LIN {X 0,Y 149.006,Z 225.633,A -85,B 0,C 180,E1 -24515.4,E2 -24515.4} C_VEL
LIN {X 0,Y 150.508,Z 227.861,A -85,B 0,C 180,E1 -24516.54,E2 -24516.54} C_VEL
LIN {X 0,Y 154.838,Z 237.074,A -85,B 0,C 180,E1 -24520.302,E2 -24520.302} C_VEL
LIN {X 0,Y 156.957,Z 243.18,A -85,B 0,C 180,E1 -24522.459,E2 -24522.459} C_VEL
LIN {X 0,Y 158.651,Z 250.853,A -85,B 0,C 180,E1 -24524.866,E2 -24524.866} C_VEL
LIN {X 0,Y 159.684,Z 260.758,A -85,B 0,C 180,E1 -24527.897,E2 -24527.897} C_VEL
LIN {X 0,Y 159.819,Z 270.245,A -85,B 0,C 180,E1 -24530.92,E2 -24530.92} C_VEL
LIN {X 0,Y 159.177,Z 278.697,A -85,B 0,C 180,E1 -24533.804,E2 -24533.804} C_VEL
LIN {X 0,Y 158.051,Z 285.315,A -85,B 0,C 180,E1 -24536.232,E2 -24536.232} C_VEL
LIN {X 0,Y 154.414,Z 293.15,A -85,B 0,C 180,E1 -24539.201,E2 -24539.201} C_VEL
LIN {X 0,Y 151.168,Z 299.693,A -85,B 0,C 180,E1 -24542.296,E2 -24542.296} C_VEL
LIN {X 0,Y 148.812,Z 304.197,A -85,B 0,C 180,E1 -24544.847,E2 -24544.847} C_VEL
LIN {X 0,Y 145.783,Z 309.692,A -85,B 0,C 180,E1 -24548.804,E2 -24548.804} C_VEL
LIN {X 0,Y 143.391,Z 314.021,A -85,B 0,C 180,E1 -24552.898,E2 -24552.898} C_VEL
LIN {X 0,Y 142.296,Z 316.395,A -85,B 0,C 180,E1 -24555.703,E2 -24555.703} C_VEL
LIN {X 0,Y 141.449,Z 318.201,A -85,B 0,C 180,E1 -24558.537,E2 -24558.537} C_VEL
LIN {X 0,Y 140.623,Z 320.663,A -85,B 0,C 180,E1 -24564.264,E2 -24564.264} C_VEL
LIN {X 0,Y 140.572,Z 321.418,A -85,B 0,C 180,E1 -24569.356,E2 -24569.356} C_VEL
LIN {X 0,Y 140.512,Z 321.259,A -85,B 0,C 180,E1 -24572.867,E2 -24572.867} C_VEL
LIN {X 0,Y 140.624,Z 320.663,A -85,B 0,C 180,E1 -24575.736,E2 -24575.736} C_VEL
LIN {X 0,Y 141.449,Z 318.201,A -85,B 0,C 180,E1 -24581.463,E2 -24581.463} C_VEL
LIN {X 0,Y 142.829,Z 315.242,A -85,B 0,C 180,E1 -24585.702,E2 -24585.702} C_VEL
LIN {X 0,Y 144.913,Z 311.247,A -85,B 0,C 180,E1 -24589.845,E2 -24589.845} C_VEL
LIN {X 0,Y 147.707,Z 306.113,A -85,B 0,C 180,E1 -24593.855,E2 -24593.855} C_VEL
LIN {X 0,Y 150.602,Z 300.85,A -85,B 0,C 180,E1 -24597.064,E2 -24597.064} C_VEL
LIN {X 0,Y 153.725,Z 294.527,A -85,B 0,C 180,E1 -24600.191,E2 -24600.191} C_VEL
LIN {X 0,Y 156.599,Z 288.573,A -85,B 0,C 180,E1 -24602.584,E2 -24602.584} C_VEL
LIN {X 0,Y 158.036,Z 285.315,A -85,B 0,C 180,E1 -24603.771,E2 -24603.771} C_VEL
LIN {X 0,Y 159.42,Z 276.844,A -85,B 0,C 180,E1 -24606.875,E2 -24606.875} C_VEL
LIN {X 0,Y 159.86,Z 266.939,A -85,B 0,C 180,E1 -24610.165,E2 -24610.165} C_VEL
LIN {X 0,Y 159.408,Z 257.125,A -85,B 0,C 180,E1 -24613.205,E2 -24613.205} C_VEL
LIN {X 0,Y 158.142,Z 248.081,A -85,B 0,C 180,E1 -24615.974,E2 -24615.974} C_VEL
LIN {X 0,Y 156.285,Z 240.912,A -85,B 0,C 180,E1 -24618.338,E2 -24618.338} C_VEL
LIN {X 0,Y 154.11,Z 235.491,A -85,B 0,C 180,E1 -24620.322,E2 -24620.322} C_VEL
LIN {X 0,Y 149.931,Z 226.822,A -85,B 0,C 180,E1 -24623.922,E2 -24623.922} C_VEL
LIN {X 0,Y 147.876,Z 223.472,A -85,B 0,C 180,E1 -24625.578,E2 -24625.578} C_VEL
LIN {X 0,Y 147.161,Z 221.537,A -85,B 0,C 180,E1 -24626.317,E2 -24626.317} C_VEL
LIN {X 0,Y 144.734,Z 218.727,A -85,B 0,C 180,E1 -24628.226,E2 -24628.226} C_VEL
LIN {X 0,Y 143.656,Z 215.787,A -85,B 0,C 180,E1 -24629.293,E2 -24629.293} C_VEL
LIN {X 0,Y 143.593,Z 215.404,A -85,B 0,C 180,E1 -24629.491,E2 -24629.491} C_VEL
LIN {X 0,Y 142.834,Z 214.884,A -85,B 0,C 180,E1 -24631.822,E2 -24631.822} C_VEL
LIN {X 0,Y 141.237,Z 214.529,A -85,B 0,C 180,E1 -24634.126,E2 -24634.126} C_VEL
LIN {X 0,Y 136.67,Z 213.808,A -85,B 0,C 180,E1 -24640.471,E2 -24640.471} C_VEL
LIN {X 0,Y 136.278,Z 213.546,A -85,B 0,C 180,E1 -24642.145,E2 -24642.145} C_VEL
LIN {X 0,Y 136.264,Z 213.03,A -85,B 0,C 180,E1 -24645.054,E2 -24645.054} C_VEL
LIN {X 0,Y 136.43,Z 212.991,A -85,B 0,C 180,E1 -24648.165,E2 -24648.165} C_VEL
LIN {X 0,Y 136.55,Z 212.976,A -85,B 0,C 180,E1 -24651.116,E2 -24651.116} C_VEL
LIN {X 0,Y 137.131,Z 212.87,A -85,B 0,C 180,E1 -24659.998,E2 -24659.998} C_VEL
LIN {X 0,Y 136.549,Z 212.968,A -85,B 0,C 180,E1 -24668.881,E2 -24668.881} C_VEL
LIN {X 0,Y 136.438,Z 212.989,A -85,B 0,C 180,E1 -24671.889,E2 -24671.889} C_VEL
LIN {X 0,Y 136.236,Z 213.014,A -85,B 0,C 180,E1 -24678.029,E2 -24678.029} C_VEL
LIN {X 0,Y 136.195,Z 213.016,A -85,B 0,C 180,E1 -24681.747,E2 -24681.747} C_VEL
LIN {X 0,Y 136.083,Z 213.063,A -85,B 0,C 180,E1 -24685.012,E2 -24685.012} C_VEL
LIN {X 0,Y 136.848,Z 215.389,A -85,B 0,C 180,E1 -24686.085,E2 -24686.085} C_VEL
LIN {X 0,Y 138.888,Z 217.815,A -85,B 0,C 180,E1 -24688.3,E2 -24688.3} C_VEL
LIN {X 0,Y 140.193,Z 218.884,A -85,B 0,C 180,E1 -24689.52,E2 -24689.52} C_VEL
LIN {X 0,Y 141.511,Z 221.601,A -85,B 0,C 180,E1 -24691.013,E2 -24691.013} C_VEL
LIN {X 0,Y 143.683,Z 223.961,A -85,B 0,C 180,E1 -24692.892,E2 -24692.892} C_VEL
LIN {X 0,Y 145.775,Z 227.545,A -85,B 0,C 180,E1 -24694.958,E2 -24694.958} C_VEL
LIN {X 0,Y 150.528,Z 235.733,A -85,B 0,C 180,E1 -24699.331,E2 -24699.331} C_VEL
LIN {X 0,Y 154.606,Z 244.364,A -85,B 0,C 180,E1 -24703.339,E2 -24703.339} C_VEL
LIN {X 0,Y 157.554,Z 252.237,A -85,B 0,C 180,E1 -24706.701,E2 -24706.701} C_VEL
LIN {X 0,Y 160.021,Z 261.291,A -85,B 0,C 180,E1 -24710.411,E2 -24710.411} C_VEL
LIN {X 0,Y 161.607,Z 270.196,A -85,B 0,C 180,E1 -24714.119,E2 -24714.119} C_VEL
LIN {X 0,Y 162.565,Z 277.467,A -85,B 0,C 180,E1 -24717.352,E2 -24717.352} C_VEL
LIN {X 0,Y 164.649,Z 285.091,A -85,B 0,C 180,E1 -24721.399,E2 -24721.399} C_VEL
LIN {X 0,Y 167.764,Z 291.175,A -85,B 0,C 180,E1 -24725.234,E2 -24725.234} C_VEL
LIN {X 0,Y 170.94,Z 295.464,A -85,B 0,C 180,E1 -24728.283,E2 -24728.283} C_VEL
LIN {X 0,Y 176.822,Z 300.472,A -85,B 0,C 180,E1 -24732.532,E2 -24732.532} C_VEL
LIN {X 0,Y 184.31,Z 304.617,A -85,B 0,C 180,E1 -24736.774,E2 -24736.774} C_VEL
LIN {X 0,Y 192.385,Z 307.533,A -85,B 0,C 180,E1 -24740.51,E2 -24740.51} C_VEL
LIN {X 0,Y 201.086,Z 309.52,A -85,B 0,C 180,E1 -24743.982,E2 -24743.982} C_VEL
LIN {X 0,Y 206.877,Z 310.378,A -85,B 0,C 180,E1 -24746.104,E2 -24746.104} C_VEL
LIN {X 0,Y 212.302,Z 310.784,A -85,B 0,C 180,E1 -24748.103,E2 -24748.103} C_VEL
LIN {X 0,Y 216.489,Z 310.826,A -85,B 0,C 180,E1 -24750,E2 -24750} C_VEL
LIN {X 0,Y 212.308,Z 310.784,A -85,B 0,C 180,E1 -24751.897,E2 -24751.897} C_VEL
LIN {X 0,Y 204.512,Z 310.094,A -85,B 0,C 180,E1 -24754.756,E2 -24754.756} C_VEL
LIN {X 0,Y 195.226,Z 308.348,A -85,B 0,C 180,E1 -24758.279,E2 -24758.279} C_VEL
LIN {X 0,Y 186.806,Z 305.664,A -85,B 0,C 180,E1 -24762,E2 -24762} C_VEL
LIN {X 0,Y 179.378,Z 302.065,A -85,B 0,C 180,E1 -24765.918,E2 -24765.918} C_VEL
LIN {X 0,Y 173.653,Z 298.041,A -85,B 0,C 180,E1 -24769.595,E2 -24769.595} C_VEL
LIN {X 0,Y 168.814,Z 292.747,A -85,B 0,C 180,E1 -24773.67,E2 -24773.67} C_VEL
LIN {X 0,Y 165.748,Z 287.634,A -85,B 0,C 180,E1 -24777.075,E2 -24777.075} C_VEL
LIN {X 0,Y 163.458,Z 281.287,A -85,B 0,C 180,E1 -24780.696,E2 -24780.696} C_VEL
LIN {X 0,Y 162.202,Z 275.384,A -85,B 0,C 180,E1 -24783.634,E2 -24783.634} C_VEL
LIN {X 0,Y 161.258,Z 267.667,A -85,B 0,C 180,E1 -24786.938,E2 -24786.938} C_VEL
LIN {X 0,Y 159.665,Z 259.89,A -85,B 0,C 180,E1 -24790.157,E2 -24790.157} C_VEL
LIN {X 0,Y 157.138,Z 251.078,A -85,B 0,C 180,E1 -24793.772,E2 -24793.772} C_VEL
LIN {X 0,Y 153.694,Z 242.257,A -85,B 0,C 180,E1 -24797.588,E2 -24797.588} C_VEL
LIN {X 0,Y 149.68,Z 234.222,A -85,B 0,C 180,E1 -24801.464,E2 -24801.464} C_VEL
LIN {X 0,Y 145.781,Z 227.545,A -85,B 0,C 180,E1 -24805.039,E2 -24805.039} C_VEL
LIN {X 0,Y 143.588,Z 223.802,A -85,B 0,C 180,E1 -24807.198,E2 -24807.198} C_VEL
LIN {X 0,Y 141.019,Z 220.798,A -85,B 0,C 180,E1 -24809.49,E2 -24809.49} C_VEL
LIN {X 0,Y 140.07,Z 218.562,A -85,B 0,C 180,E1 -24810.639,E2 -24810.639} C_VEL
LIN {X 0,Y 137.435,Z 216.322,A -85,B 0,C 180,E1 -24813.217,E2 -24813.217} C_VEL
LIN {X 0,Y 136.309,Z 214.128,A -85,B 0,C 180,E1 -24814.624,E2 -24814.624} C_VEL
LIN {X 0,Y 136.084,Z 213.023,A -85,B 0,C 180,E1 -24815.09,E2 -24815.09} C_VEL
LIN {X 0,Y 136.241,Z 213.007,A -85,B 0,C 180,E1 -24818.834,E2 -24818.834} C_VEL
LIN {X 0,Y 136.262,Z 213.001,A -85,B 0,C 180,E1 -24825.057,E2 -24825.057} C_VEL
LIN {X 0,Y 136.429,Z 212.99,A -85,B 0,C 180,E1 -24828.167,E2 -24828.167} C_VEL
LIN {X 0,Y 136.549,Z 212.968,A -85,B 0,C 180,E1 -24831.119,E2 -24831.119} C_VEL
LIN {X 0,Y 137.131,Z 212.87,A -85,B 0,C 180,E1 -24840.002,E2 -24840.002} C_VEL
LIN {X 0,Y 136.55,Z 212.976,A -85,B 0,C 180,E1 -24848.884,E2 -24848.884} C_VEL
LIN {X 0,Y 136.44,Z 212.992,A -85,B 0,C 180,E1 -24851.892,E2 -24851.892} C_VEL
LIN {X 0,Y 136.264,Z 213.031,A -85,B 0,C 180,E1 -24854.946,E2 -24854.946} C_VEL
LIN {X 0,Y 136.387,Z 214.204,A -85,B 0,C 180,E1 -24861.145,E2 -24861.145} C_VEL
LIN {X 0,Y 136.394,Z 215.177,A -85,B 0,C 180,E1 -24865.057,E2 -24865.057} C_VEL
LIN {X 0,Y 137.554,Z 218.297,A -85,B 0,C 180,E1 -24866.557,E2 -24866.557} C_VEL
LIN {X 0,Y 140.111,Z 221.359,A -85,B 0,C 180,E1 -24869.122,E2 -24869.122} C_VEL
LIN {X 0,Y 140.608,Z 222.147,A -85,B 0,C 180,E1 -24869.639,E2 -24869.639} C_VEL
LIN {X 0,Y 142.086,Z 225.426,A -85,B 0,C 180,E1 -24871.291,E2 -24871.291} C_VEL
LIN {X 0,Y 143.909,Z 227.957,A -85,B 0,C 180,E1 -24872.911,E2 -24872.911} C_VEL
LIN {X 0,Y 145.536,Z 231.425,A -85,B 0,C 180,E1 -24874.572,E2 -24874.572} C_VEL
LIN {X 0,Y 146.29,Z 232.543,A -85,B 0,C 180,E1 -24875.245,E2 -24875.245} C_VEL
LIN {X 0,Y 150.351,Z 242.131,A -85,B 0,C 180,E1 -24879.437,E2 -24879.437} C_VEL
LIN {X 0,Y 152.318,Z 249.001,A -85,B 0,C 180,E1 -24881.996,E2 -24881.996} C_VEL
LIN {X 0,Y 153.315,Z 256.047,A -85,B 0,C 180,E1 -24884.384,E2 -24884.384} C_VEL
LIN {X 0,Y 153.814,Z 263.83,A -85,B 0,C 180,E1 -24886.978,E2 -24886.978} C_VEL
LIN {X 0,Y 153.711,Z 271.366,A -85,B 0,C 180,E1 -24889.554,E2 -24889.554} C_VEL
LIN {X 0,Y 153.004,Z 279.042,A -85,B 0,C 180,E1 -24892.339,E2 -24892.339} C_VEL
LIN {X 0,Y 151.946,Z 285.095,A -85,B 0,C 180,E1 -24894.679,E2 -24894.679} C_VEL
LIN {X 0,Y 150.671,Z 288.362,A -85,B 0,C 180,E1 -24895.963,E2 -24895.963} C_VEL
LIN {X 0,Y 147.603,Z 294.315,A -85,B 0,C 180,E1 -24898.416,E2 -24898.416} C_VEL
LIN {X 0,Y 144.259,Z 300.637,A -85,B 0,C 180,E1 -24901.641,E2 -24901.641} C_VEL
LIN {X 0,Y 141.211,Z 305.9,A -85,B 0,C 180,E1 -24904.974,E2 -24904.974} C_VEL
LIN {X 0,Y 138.218,Z 311.034,A -85,B 0,C 180,E1 -24909.15,E2 -24909.15} C_VEL
LIN {X 0,Y 135.96,Z 315.029,A -85,B 0,C 180,E1 -24913.483,E2 -24913.483} C_VEL
LIN {X 0,Y 134.481,Z 317.989,A -85,B 0,C 180,E1 -24917.934,E2 -24917.934} C_VEL
LIN {X 0,Y 133.55,Z 320.452,A -85,B 0,C 180,E1 -24923.959,E2 -24923.959} C_VEL
LIN {X 0,Y 133.415,Z 321.047,A -85,B 0,C 180,E1 -24926.98,E2 -24926.98} C_VEL
LIN {X 0,Y 133.535,Z 321.209,A -85,B 0,C 180,E1 -24930,E2 -24930} C_VEL
LIN {X 0,Y 133.415,Z 321.047,A -85,B 0,C 180,E1 -24933.02,E2 -24933.02} C_VEL
LIN {X 0,Y 133.55,Z 320.452,A -85,B 0,C 180,E1 -24936.041,E2 -24936.041} C_VEL
LIN {X 0,Y 134.481,Z 317.989,A -85,B 0,C 180,E1 -24942.066,E2 -24942.066} C_VEL
LIN {X 0,Y 135.96,Z 315.029,A -85,B 0,C 180,E1 -24946.517,E2 -24946.517} C_VEL
LIN {X 0,Y 138.218,Z 311.034,A -85,B 0,C 180,E1 -24950.85,E2 -24950.85} C_VEL
LIN {X 0,Y 141.213,Z 305.9,A -85,B 0,C 180,E1 -24955.026,E2 -24955.026} C_VEL
LIN {X 0,Y 144.278,Z 300.638,A -85,B 0,C 180,E1 -24958.355,E2 -24958.355} C_VEL
LIN {X 0,Y 146.807,Z 295.829,A -85,B 0,C 180,E1 -24960.892,E2 -24960.892} C_VEL
LIN {X 0,Y 149.855,Z 289.989,A -85,B 0,C 180,E1 -24963.439,E2 -24963.439} C_VEL
LIN {X 0,Y 151.976,Z 285.096,A -85,B 0,C 180,E1 -24965.313,E2 -24965.313} C_VEL
LIN {X 0,Y 153.419,Z 275.912,A -85,B 0,C 180,E1 -24968.851,E2 -24968.851} C_VEL
LIN {X 0,Y 153.842,Z 265.789,A -85,B 0,C 180,E1 -24972.378,E2 -24972.378} C_VEL
LIN {X 0,Y 153.465,Z 257.36,A -85,B 0,C 180,E1 -24975.191,E2 -24975.191} C_VEL
LIN {X 0,Y 152.318,Z 249,A -85,B 0,C 180,E1 -24978.004,E2 -24978.004} C_VEL
LIN {X 0,Y 150.359,Z 242.108,A -85,B 0,C 180,E1 -24980.565,E2 -24980.565} C_VEL
LIN {X 0,Y 146.267,Z 232.458,A -85,B 0,C 180,E1 -24984.787,E2 -24984.787} C_VEL
LIN {X 0,Y 144.221,Z 228.779,A -85,B 0,C 180,E1 -24986.753,E2 -24986.753} C_VEL
LIN {X 0,Y 143.289,Z 226.926,A -85,B 0,C 180,E1 -24987.659,E2 -24987.659} C_VEL
LIN {X 0,Y 141.184,Z 223.799,A -85,B 0,C 180,E1 -24989.629,E2 -24989.629} C_VEL
LIN {X 0,Y 140.238,Z 221.36,A -85,B 0,C 180,E1 -24990.786,E2 -24990.786} C_VEL
LIN {X 0,Y 137.633,Z 218.428,A -85,B 0,C 180,E1 -24993.357,E2 -24993.357} C_VEL
LIN {X 0,Y 136.433,Z 215.428,A -85,B 0,C 180,E1 -24994.849,E2 -24994.849} C_VEL
LIN {X 0,Y 136.356,Z 214.979,A -85,B 0,C 180,E1 -24995.241,E2 -24995.241} C_VEL
LIN {X 0,Y 136.369,Z 214.185,A -85,B 0,C 180,E1 -24998.852,E2 -24998.852} C_VEL
LIN {X 0,Y 136.278,Z 213.546,A -85,B 0,C 180,E1 -25002.145,E2 -25002.145} C_VEL
LIN {X 0,Y 135.512,Z 213.301,A -85,B 0,C 180,E1 -25004.613,E2 -25004.613} C_VEL
LIN {X 0,Y 133.935,Z 213.342,A -85,B 0,C 180,E1 -25007.055,E2 -25007.055} C_VEL
LIN {X 0,Y 129.732,Z 213.826,A -85,B 0,C 180,E1 -25013.797,E2 -25013.797} C_VEL
LIN {X 0,Y 129.544,Z 213.843,A -85,B 0,C 180,E1 -25015.569,E2 -25015.569} C_VEL
LIN {X 0,Y 130.086,Z 213.745,A -85,B 0,C 180,E1 -25019.998,E2 -25019.998} C_VEL
LIN {X 0,Y 129.472,Z 213.847,A -85,B 0,C 180,E1 -25029.37,E2 -25029.37} C_VEL
LIN {X 0,Y 129.342,Z 213.874,A -85,B 0,C 180,E1 -25032.551,E2 -25032.551} C_VEL
LIN {X 0,Y 129.181,Z 213.97,A -85,B 0,C 180,E1 -25037.409,E2 -25037.409} C_VEL
LIN {X 0,Y 129.981,Z 216.424,A -85,B 0,C 180,E1 -25039.133,E2 -25039.133} C_VEL
LIN {X 0,Y 132.512,Z 219.142,A -85,B 0,C 180,E1 -25042.909,E2 -25042.909} C_VEL
LIN {X 0,Y 133.419,Z 219.722,A -85,B 0,C 180,E1 -25043.989,E2 -25043.989} C_VEL
LIN {X 0,Y 134.691,Z 222.539,A -85,B 0,C 180,E1 -25045.911,E2 -25045.911} C_VEL
LIN {X 0,Y 136.26,Z 224.238,A -85,B 0,C 180,E1 -25047.657,E2 -25047.657} C_VEL
LIN {X 0,Y 138.601,Z 227.97,A -85,B 0,C 180,E1 -25050.467,E2 -25050.467} C_VEL
LIN {X 0,Y 139.95,Z 229.469,A -85,B 0,C 180,E1 -25051.821,E2 -25051.821} C_VEL
LIN {X 0,Y 144.323,Z 237.375,A -85,B 0,C 180,E1 -25056.62,E2 -25056.62} C_VEL
LIN {X 0,Y 147.84,Z 244.665,A -85,B 0,C 180,E1 -25060.484,E2 -25060.484} C_VEL
LIN {X 0,Y 150.929,Z 252.576,A -85,B 0,C 180,E1 -25064.303,E2 -25064.303} C_VEL
LIN {X 0,Y 153.311,Z 261.085,A -85,B 0,C 180,E1 -25068.133,E2 -25068.133} C_VEL
LIN {X 0,Y 154.975,Z 269.893,A -85,B 0,C 180,E1 -25072.084,E2 -25072.084} C_VEL
LIN {X 0,Y 155.816,Z 278.256,A -85,B 0,C 180,E1 -25076.017,E2 -25076.017} C_VEL
LIN {X 0,Y 157.268,Z 285.343,A -85,B 0,C 180,E1 -25079.922,E2 -25079.922} C_VEL
LIN {X 0,Y 159.768,Z 291.439,A -85,B 0,C 180,E1 -25083.904,E2 -25083.904} C_VEL
LIN {X 0,Y 164.081,Z 297.332,A -85,B 0,C 180,E1 -25088.5,E2 -25088.5} C_VEL
LIN {X 0,Y 167.943,Z 300.771,A -85,B 0,C 180,E1 -25091.598,E2 -25091.598} C_VEL
LIN {X 0,Y 174.956,Z 304.897,A -85,B 0,C 180,E1 -25096.053,E2 -25096.053} C_VEL
LIN {X 0,Y 180.175,Z 307.032,A -85,B 0,C 180,E1 -25098.754,E2 -25098.754} C_VEL
LIN {X 0,Y 190.984,Z 309.722,A -85,B 0,C 180,E1 -25103.487,E2 -25103.487} C_VEL
LIN {X 0,Y 197.409,Z 310.658,A -85,B 0,C 180,E1 -25105.917,E2 -25105.917} C_VEL
LIN {X 0,Y 203.9,Z 311.099,A -85,B 0,C 180,E1 -25108.279,E2 -25108.279} C_VEL
LIN {X 0,Y 208.184,Z 311.069,A -85,B 0,C 180,E1 -25110,E2 -25110} C_VEL
LIN {X 0,Y 203.179,Z 311.054,A -85,B 0,C 180,E1 -25111.982,E2 -25111.982} C_VEL
LIN {X 0,Y 197.29,Z 310.649,A -85,B 0,C 180,E1 -25114.123,E2 -25114.123} C_VEL
LIN {X 0,Y 184.998,Z 308.449,A -85,B 0,C 180,E1 -25118.993,E2 -25118.993} C_VEL
LIN {X 0,Y 179.38,Z 306.765,A -85,B 0,C 180,E1 -25121.632,E2 -25121.632} C_VEL
LIN {X 0,Y 172.478,Z 303.671,A -85,B 0,C 180,E1 -25125.438,E2 -25125.438} C_VEL
LIN {X 0,Y 166.105,Z 299.346,A -85,B 0,C 180,E1 -25129.784,E2 -25129.784} C_VEL
LIN {X 0,Y 161.561,Z 294.291,A -85,B 0,C 180,E1 -25134.008,E2 -25134.008} C_VEL
LIN {X 0,Y 158.349,Z 288.374,A -85,B 0,C 180,E1 -25138.188,E2 -25138.188} C_VEL
LIN {X 0,Y 156.396,Z 281.808,A -85,B 0,C 180,E1 -25142.112,E2 -25142.112} C_VEL
LIN {X 0,Y 155.481,Z 275.03,A -85,B 0,C 180,E1 -25145.551,E2 -25145.551} C_VEL
LIN {X 0,Y 154.79,Z 268.616,A -85,B 0,C 180,E1 -25148.494,E2 -25148.494} C_VEL
LIN {X 0,Y 152.839,Z 259.326,A -85,B 0,C 180,E1 -25152.633,E2 -25152.633} C_VEL
LIN {X 0,Y 150.408,Z 251.155,A -85,B 0,C 180,E1 -25156.344,E2 -25156.344} C_VEL
LIN {X 0,Y 147.826,Z 244.666,A -85,B 0,C 180,E1 -25159.523,E2 -25159.523} C_VEL
LIN {X 0,Y 144.31,Z 237.414,A -85,B 0,C 180,E1 -25163.376,E2 -25163.376} C_VEL
LIN {X 0,Y 139.956,Z 229.446,A -85,B 0,C 180,E1 -25168.181,E2 -25168.181} C_VEL
LIN {X 0,Y 138.561,Z 227.942,A -85,B 0,C 180,E1 -25169.57,E2 -25169.57} C_VEL
LIN {X 0,Y 136.096,Z 224.073,A -85,B 0,C 180,E1 -25172.516,E2 -25172.516} C_VEL
LIN {X 0,Y 134.021,Z 221.394,A -85,B 0,C 180,E1 -25174.991,E2 -25174.991} C_VEL
LIN {X 0,Y 133.205,Z 219.513,A -85,B 0,C 180,E1 -25176.28,E2 -25176.28} C_VEL
LIN {X 0,Y 130.512,Z 217.267,A -85,B 0,C 180,E1 -25179.924,E2 -25179.924} C_VEL
LIN {X 0,Y 129.377,Z 214.877,A -85,B 0,C 180,E1 -25182.108,E2 -25182.108} C_VEL
LIN {X 0,Y 129.175,Z 213.895,A -85,B 0,C 180,E1 -25182.794,E2 -25182.794} C_VEL
LIN {X 0,Y 129.374,Z 213.87,A -85,B 0,C 180,E1 -25187.905,E2 -25187.905} C_VEL
LIN {X 0,Y 129.472,Z 213.847,A -85,B 0,C 180,E1 -25190.63,E2 -25190.63} C_VEL
LIN {X 0,Y 130.086,Z 213.745,A -85,B 0,C 180,E1 -25200.002,E2 -25200.002} C_VEL
LIN {X 0,Y 129.473,Z 213.859,A -85,B 0,C 180,E1 -25209.374,E2 -25209.374} C_VEL
LIN {X 0,Y 129.343,Z 213.875,A -85,B 0,C 180,E1 -25212.555,E2 -25212.555} C_VEL
LIN {X 0,Y 129.267,Z 214.62,A -85,B 0,C 180,E1 -25217.095,E2 -25217.095} C_VEL
LIN {X 0,Y 130.359,Z 217.723,A -85,B 0,C 180,E1 -25219.284,E2 -25219.284} C_VEL
LIN {X 0,Y 133.213,Z 221.135,A -85,B 0,C 180,E1 -25223.31,E2 -25223.31} C_VEL
LIN {X 0,Y 133.782,Z 221.779,A -85,B 0,C 180,E1 -25224.027,E2 -25224.027} C_VEL
LIN {X 0,Y 135.19,Z 225.149,A -85,B 0,C 180,E1 -25226.122,E2 -25226.122} C_VEL
LIN {X 0,Y 137.4,Z 228.079,A -85,B 0,C 180,E1 -25228.552,E2 -25228.552} C_VEL
LIN {X 0,Y 138.838,Z 231.362,A -85,B 0,C 180,E1 -25230.413,E2 -25230.413} C_VEL
LIN {X 0,Y 140.007,Z 233.031,A -85,B 0,C 180,E1 -25231.641,E2 -25231.641} C_VEL
LIN {X 0,Y 141.23,Z 236.091,A -85,B 0,C 180,E1 -25233.19,E2 -25233.19} C_VEL
LIN {X 0,Y 142.565,Z 238.665,A -85,B 0,C 180,E1 -25234.602,E2 -25234.602} C_VEL
LIN {X 0,Y 145.846,Z 247.591,A -85,B 0,C 180,E1 -25238.79,E2 -25238.79} C_VEL
LIN {X 0,Y 147.048,Z 252.739,A -85,B 0,C 180,E1 -25240.881,E2 -25240.881} C_VEL
LIN {X 0,Y 147.835,Z 260.613,A -85,B 0,C 180,E1 -25243.721,E2 -25243.721} C_VEL
LIN {X 0,Y 147.836,Z 270.041,A -85,B 0,C 180,E1 -25247.146,E2 -25247.146} C_VEL
LIN {X 0,Y 147.265,Z 277.037,A -85,B 0,C 180,E1 -25249.782,E2 -25249.782} C_VEL
LIN {X 0,Y 145.904,Z 284.872,A -85,B 0,C 180,E1 -25252.98,E2 -25252.98} C_VEL
LIN {X 0,Y 144.796,Z 288.149,A -85,B 0,C 180,E1 -25254.378,E2 -25254.378} C_VEL
LIN {X 0,Y 141.572,Z 294.102,A -85,B 0,C 180,E1 -25256.903,E2 -25256.903} C_VEL
LIN {X 0,Y 138.146,Z 300.153,A -85,B 0,C 180,E1 -25260.067,E2 -25260.067} C_VEL
LIN {X 0,Y 136.084,Z 303.774,A -85,B 0,C 180,E1 -25262.303,E2 -25262.303} C_VEL
LIN {X 0,Y 132.592,Z 309.267,A -85,B 0,C 180,E1 -25266.576,E2 -25266.576} C_VEL
LIN {X 0,Y 129.819,Z 313.596,A -85,B 0,C 180,E1 -25271.046,E2 -25271.046} C_VEL
LIN {X 0,Y 128.537,Z 315.971,A -85,B 0,C 180,E1 -25274.135,E2 -25274.135} C_VEL
LIN {X 0,Y 127.509,Z 317.777,A -85,B 0,C 180,E1 -25277.264,E2 -25277.264} C_VEL
LIN {X 0,Y 126.471,Z 320.24,A -85,B 0,C 180,E1 -25283.619,E2 -25283.619} C_VEL
LIN {X 0,Y 126.318,Z 320.836,A -85,B 0,C 180,E1 -25286.811,E2 -25286.811} C_VEL
LIN {X 0,Y 126.449,Z 320.998,A -85,B 0,C 180,E1 -25290,E2 -25290} C_VEL
LIN {X 0,Y 126.318,Z 320.836,A -85,B 0,C 180,E1 -25293.189,E2 -25293.189} C_VEL
LIN {X 0,Y 126.471,Z 320.24,A -85,B 0,C 180,E1 -25296.381,E2 -25296.381} C_VEL
LIN {X 0,Y 127.51,Z 317.777,A -85,B 0,C 180,E1 -25302.736,E2 -25302.736} C_VEL
LIN {X 0,Y 129.133,Z 314.817,A -85,B 0,C 180,E1 -25307.417,E2 -25307.417} C_VEL
LIN {X 0,Y 131.578,Z 310.822,A -85,B 0,C 180,E1 -25311.956,E2 -25311.956} C_VEL
LIN {X 0,Y 134.793,Z 305.689,A -85,B 0,C 180,E1 -25316.307,E2 -25316.307} C_VEL
LIN {X 0,Y 137.378,Z 301.582,A -85,B 0,C 180,E1 -25319.078,E2 -25319.078} C_VEL
LIN {X 0,Y 140.728,Z 295.616,A -85,B 0,C 180,E1 -25322.385,E2 -25322.385} C_VEL
LIN {X 0,Y 143.95,Z 289.776,A -85,B 0,C 180,E1 -25325.005,E2 -25325.005} C_VEL
LIN {X 0,Y 145.473,Z 286.516,A -85,B 0,C 180,E1 -25326.285,E2 -25326.285} C_VEL
LIN {X 0,Y 147.011,Z 278.771,A -85,B 0,C 180,E1 -25329.506,E2 -25329.506} C_VEL
LIN {X 0,Y 147.715,Z 271.455,A -85,B 0,C 180,E1 -25332.328,E2 -25332.328} C_VEL
LIN {X 0,Y 147.92,Z 263.51,A -85,B 0,C 180,E1 -25335.218,E2 -25335.218} C_VEL
LIN {X 0,Y 147.565,Z 256.846,A -85,B 0,C 180,E1 -25337.625,E2 -25337.625} C_VEL
LIN {X 0,Y 146.592,Z 250.321,A -85,B 0,C 180,E1 -25340.092,E2 -25340.092} C_VEL
LIN {X 0,Y 144.753,Z 244.363,A -85,B 0,C 180,E1 -25342.633,E2 -25342.633} C_VEL
LIN {X 0,Y 142.169,Z 237.661,A -85,B 0,C 180,E1 -25345.867,E2 -25345.867} C_VEL
LIN {X 0,Y 140.581,Z 234.649,A -85,B 0,C 180,E1 -25347.575,E2 -25347.575} C_VEL
LIN {X 0,Y 140.022,Z 232.981,A -85,B 0,C 180,E1 -25348.363,E2 -25348.363} C_VEL
LIN {X 0,Y 138.264,Z 230.273,A -85,B 0,C 180,E1 -25350.289,E2 -25350.289} C_VEL
LIN {X 0,Y 137.035,Z 227.344,A -85,B 0,C 180,E1 -25351.887,E2 -25351.887} C_VEL
LIN {X 0,Y 134.638,Z 224.157,A -85,B 0,C 180,E1 -25354.593,E2 -25354.593} C_VEL
LIN {X 0,Y 133.537,Z 221.273,A -85,B 0,C 180,E1 -25356.339,E2 -25356.339} C_VEL
LIN {X 0,Y 130.586,Z 218.143,A -85,B 0,C 180,E1 -25360.342,E2 -25360.342} C_VEL
LIN {X 0,Y 129.367,Z 215.104,A -85,B 0,C 180,E1 -25362.613,E2 -25362.613} C_VEL
LIN {X 0,Y 129.233,Z 214.522,A -85,B 0,C 180,E1 -25363.002,E2 -25363.002} C_VEL
LIN {X 0,Y 129.375,Z 213.87,A -85,B 0,C 180,E1 -25367.902,E2 -25367.902} C_VEL
LIN {X 0,Y 129.473,Z 213.859,A -85,B 0,C 180,E1 -25370.626,E2 -25370.626} C_VEL
LIN {X 0,Y 129.544,Z 213.843,A -85,B 0,C 180,E1 -25375.569,E2 -25375.569} C_VEL
LIN {X 0,Y 129.049,Z 214.12,A -85,B 0,C 180,E1 -25378.164,E2 -25378.164} C_VEL
LIN {X 0,Y 127.66,Z 214.851,A -85,B 0,C 180,E1 -25380.723,E2 -25380.723} C_VEL
LIN {X 0,Y 124.549,Z 217.043,A -85,B 0,C 180,E1 -25385.931,E2 -25385.931} C_VEL
LIN {X 0,Y 124.024,Z 218.212,A -85,B 0,C 180,E1 -25388.646,E2 -25388.646} C_VEL
LIN {X 0,Y 124.157,Z 218.575,A -85,B 0,C 180,E1 -25389.556,E2 -25389.556} C_VEL
LIN {X 0,Y 127.018,Z 220.87,A -85,B 0,C 180,E1 -25396.575,E2 -25396.575} C_VEL
LIN {X 0,Y 128.03,Z 223.489,A -85,B 0,C 180,E1 -25399.02,E2 -25399.02} C_VEL
LIN {X 0,Y 130.09,Z 225.65,A -85,B 0,C 180,E1 -25402.218,E2 -25402.218} C_VEL
LIN {X 0,Y 134.08,Z 231.807,A -85,B 0,C 180,E1 -25408.146,E2 -25408.146} C_VEL
LIN {X 0,Y 136.41,Z 235.342,A -85,B 0,C 180,E1 -25411.01,E2 -25411.01} C_VEL
LIN {X 0,Y 140.812,Z 244.388,A -85,B 0,C 180,E1 -25416.791,E2 -25416.791} C_VEL
LIN {X 0,Y 143.686,Z 251.347,A -85,B 0,C 180,E1 -25420.734,E2 -25420.734} C_VEL
LIN {X 0,Y 145.907,Z 258.241,A -85,B 0,C 180,E1 -25424.297,E2 -25424.297} C_VEL
LIN {X 0,Y 147.456,Z 264.637,A -85,B 0,C 180,E1 -25427.443,E2 -25427.443} C_VEL
LIN {X 0,Y 148.633,Z 271.99,A -85,B 0,C 180,E1 -25431.023,E2 -25431.023} C_VEL
LIN {X 0,Y 149.134,Z 278.252,A -85,B 0,C 180,E1 -25434.139,E2 -25434.139} C_VEL
LIN {X 0,Y 150.084,Z 285.559,A -85,B 0,C 180,E1 -25438.301,E2 -25438.301} C_VEL
LIN {X 0,Y 152.076,Z 291.695,A -85,B 0,C 180,E1 -25442.475,E2 -25442.475} C_VEL
LIN {X 0,Y 154.536,Z 295.991,A -85,B 0,C 180,E1 -25445.839,E2 -25445.839} C_VEL
LIN {X 0,Y 159.436,Z 301.252,A -85,B 0,C 180,E1 -25450.769,E2 -25450.769} C_VEL
LIN {X 0,Y 165.777,Z 305.174,A -85,B 0,C 180,E1 -25455.264,E2 -25455.264} C_VEL
LIN {X 0,Y 171.955,Z 307.707,A -85,B 0,C 180,E1 -25458.779,E2 -25458.779} C_VEL
LIN {X 0,Y 177.642,Z 309.315,A -85,B 0,C 180,E1 -25461.512,E2 -25461.512} C_VEL
LIN {X 0,Y 187.765,Z 310.943,A -85,B 0,C 180,E1 -25465.707,E2 -25465.707} C_VEL
LIN {X 0,Y 196.81,Z 311.397,A -85,B 0,C 180,E1 -25468.99,E2 -25468.99} C_VEL
LIN {X 0,Y 199.463,Z 311.324,A -85,B 0,C 180,E1 -25470,E2 -25470} C_VEL
LIN {X 0,Y 193.785,Z 311.333,A -85,B 0,C 180,E1 -25472.078,E2 -25472.078} C_VEL
LIN {X 0,Y 183.686,Z 310.411,A -85,B 0,C 180,E1 -25475.866,E2 -25475.866} C_VEL
LIN {X 0,Y 176.1,Z 308.913,A -85,B 0,C 180,E1 -25479.186,E2 -25479.186} C_VEL
LIN {X 0,Y 170.708,Z 307.32,A -85,B 0,C 180,E1 -25481.879,E2 -25481.879} C_VEL
LIN {X 0,Y 161.945,Z 303.035,A -85,B 0,C 180,E1 -25487.308,E2 -25487.308} C_VEL
LIN {X 0,Y 157.602,Z 299.615,A -85,B 0,C 180,E1 -25490.9,E2 -25490.9} C_VEL
LIN {X 0,Y 153.178,Z 293.908,A -85,B 0,C 180,E1 -25495.839,E2 -25495.839} C_VEL
LIN {X 0,Y 150.691,Z 288.005,A -85,B 0,C 180,E1 -25500.122,E2 -25500.122} C_VEL
LIN {X 0,Y 149.312,Z 280.979,A -85,B 0,C 180,E1 -25504.39,E2 -25504.39} C_VEL
LIN {X 0,Y 148.859,Z 274.249,A -85,B 0,C 180,E1 -25507.861,E2 -25507.861} C_VEL
LIN {X 0,Y 147.916,Z 267.193,A -85,B 0,C 180,E1 -25511.332,E2 -25511.332} C_VEL
LIN {X 0,Y 146.344,Z 259.918,A -85,B 0,C 180,E1 -25514.902,E2 -25514.902} C_VEL
LIN {X 0,Y 144.364,Z 253.129,A -85,B 0,C 180,E1 -25518.34,E2 -25518.34} C_VEL
LIN {X 0,Y 141.101,Z 244.985,A -85,B 0,C 180,E1 -25522.837,E2 -25522.837} C_VEL
LIN {X 0,Y 137.961,Z 238.6,A -85,B 0,C 180,E1 -25526.798,E2 -25526.798} C_VEL
LIN {X 0,Y 136.413,Z 235.332,A -85,B 0,C 180,E1 -25528.991,E2 -25528.991} C_VEL
LIN {X 0,Y 132.976,Z 230.213,A -85,B 0,C 180,E1 -25533.307,E2 -25533.307} C_VEL
LIN {X 0,Y 129.819,Z 225.447,A -85,B 0,C 180,E1 -25538.151,E2 -25538.151} C_VEL
LIN {X 0,Y 127.551,Z 222.634,A -85,B 0,C 180,E1 -25541.947,E2 -25541.947} C_VEL
LIN {X 0,Y 126.986,Z 220.749,A -85,B 0,C 180,E1 -25543.524,E2 -25543.524} C_VEL
LIN {X 0,Y 123.204,Z 215.54,A -85,B 0,C 180,E1 -25560.002,E2 -25560.002} C_VEL
LIN {X 0,Y 125.057,Z 219.479,A -85,B 0,C 180,E1 -25571.497,E2 -25571.497} C_VEL
LIN {X 0,Y 127.156,Z 221.411,A -85,B 0,C 180,E1 -25576.147,E2 -25576.147} C_VEL
LIN {X 0,Y 128.336,Z 224.698,A -85,B 0,C 180,E1 -25578.977,E2 -25578.977} C_VEL
LIN {X 0,Y 131.002,Z 228.036,A -85,B 0,C 180,E1 -25582.995,E2 -25582.995} C_VEL
LIN {X 0,Y 132.207,Z 231.177,A -85,B 0,C 180,E1 -25585.17,E2 -25585.17} C_VEL
LIN {X 0,Y 133.853,Z 233.572,A -85,B 0,C 180,E1 -25587.351,E2 -25587.351} C_VEL
LIN {X 0,Y 135.334,Z 237.164,A -85,B 0,C 180,E1 -25589.562,E2 -25589.562} C_VEL
LIN {X 0,Y 138.01,Z 242.974,A -85,B 0,C 180,E1 -25593.193,E2 -25593.193} C_VEL
LIN {X 0,Y 140.479,Z 250.222,A -85,B 0,C 180,E1 -25596.896,E2 -25596.896} C_VEL
LIN {X 0,Y 141.766,Z 256.364,A -85,B 0,C 180,E1 -25599.665,E2 -25599.665} C_VEL
LIN {X 0,Y 142.152,Z 262.595,A -85,B 0,C 180,E1 -25602.133,E2 -25602.133} C_VEL
LIN {X 0,Y 142.012,Z 269.967,A -85,B 0,C 180,E1 -25604.999,E2 -25604.999} C_VEL
LIN {X 0,Y 141.203,Z 278.082,A -85,B 0,C 180,E1 -25608.298,E2 -25608.298} C_VEL
LIN {X 0,Y 139.919,Z 284.646,A -85,B 0,C 180,E1 -25611.108,E2 -25611.108} C_VEL
LIN {X 0,Y 138.976,Z 287.934,A -85,B 0,C 180,E1 -25612.64,E2 -25612.64} C_VEL
LIN {X 0,Y 135.643,Z 293.89,A -85,B 0,C 180,E1 -25615.255,E2 -25615.255} C_VEL
LIN {X 0,Y 131.621,Z 300.55,A -85,B 0,C 180,E1 -25618.89,E2 -25618.89} C_VEL
LIN {X 0,Y 128.45,Z 305.477,A -85,B 0,C 180,E1 -25622.286,E2 -25622.286} C_VEL
LIN {X 0,Y 124.997,Z 310.61,A -85,B 0,C 180,E1 -25626.823,E2 -25626.823} C_VEL
LIN {X 0,Y 122.327,Z 314.604,A -85,B 0,C 180,E1 -25631.58,E2 -25631.58} C_VEL
LIN {X 0,Y 120.569,Z 317.565,A -85,B 0,C 180,E1 -25636.517,E2 -25636.517} C_VEL
LIN {X 0,Y 119.417,Z 320.029,A -85,B 0,C 180,E1 -25643.24,E2 -25643.24} C_VEL
LIN {X 0,Y 119.232,Z 320.625,A -85,B 0,C 180,E1 -25646.621,E2 -25646.621} C_VEL
LIN {X 0,Y 119.364,Z 320.787,A -85,B 0,C 180,E1 -25650,E2 -25650} C_VEL
LIN {X 0,Y 119.232,Z 320.625,A -85,B 0,C 180,E1 -25653.379,E2 -25653.379} C_VEL
LIN {X 0,Y 119.417,Z 320.029,A -85,B 0,C 180,E1 -25656.76,E2 -25656.76} C_VEL
LIN {X 0,Y 120.569,Z 317.565,A -85,B 0,C 180,E1 -25663.483,E2 -25663.483} C_VEL
LIN {X 0,Y 122.327,Z 314.604,A -85,B 0,C 180,E1 -25668.42,E2 -25668.42} C_VEL
LIN {X 0,Y 124.997,Z 310.61,A -85,B 0,C 180,E1 -25673.177,E2 -25673.177} C_VEL
LIN {X 0,Y 128.453,Z 305.477,A -85,B 0,C 180,E1 -25677.713,E2 -25677.713} C_VEL
LIN {X 0,Y 131.669,Z 300.488,A -85,B 0,C 180,E1 -25681.146,E2 -25681.146} C_VEL
LIN {X 0,Y 135.626,Z 293.889,A -85,B 0,C 180,E1 -25684.75,E2 -25684.75} C_VEL
LIN {X 0,Y 138.977,Z 287.934,A -85,B 0,C 180,E1 -25687.36,E2 -25687.36} C_VEL
LIN {X 0,Y 140.701,Z 280.931,A -85,B 0,C 180,E1 -25690.492,E2 -25690.492} C_VEL
LIN {X 0,Y 141.635,Z 274.603,A -85,B 0,C 180,E1 -25693.162,E2 -25693.162} C_VEL
LIN {X 0,Y 142.222,Z 265.603,A -85,B 0,C 180,E1 -25696.697,E2 -25696.697} C_VEL
LIN {X 0,Y 141.93,Z 257.356,A -85,B 0,C 180,E1 -25699.928,E2 -25699.928} C_VEL
LIN {X 0,Y 140.894,Z 251.787,A -85,B 0,C 180,E1 -25702.333,E2 -25702.333} C_VEL
LIN {X 0,Y 138.48,Z 244.405,A -85,B 0,C 180,E1 -25706.063,E2 -25706.063} C_VEL
LIN {X 0,Y 135.945,Z 238.115,A -85,B 0,C 180,E1 -25709.73,E2 -25709.73} C_VEL
LIN {X 0,Y 134.286,Z 234.899,A -85,B 0,C 180,E1 -25711.897,E2 -25711.897} C_VEL
LIN {X 0,Y 133.846,Z 233.594,A -85,B 0,C 180,E1 -25712.648,E2 -25712.648} C_VEL
LIN {X 0,Y 131.745,Z 230.238,A -85,B 0,C 180,E1 -25715.578,E2 -25715.578} C_VEL
LIN {X 0,Y 130.698,Z 227.484,A -85,B 0,C 180,E1 -25717.47,E2 -25717.47} C_VEL
LIN {X 0,Y 127.941,Z 223.952,A -85,B 0,C 180,E1 -25721.793,E2 -25721.793} C_VEL
LIN {X 0,Y 127.044,Z 221.105,A -85,B 0,C 180,E1 -25724.147,E2 -25724.147} C_VEL
LIN {X 0,Y 123.184,Z 215.622,A -85,B 0,C 180,E1 -25739.794,E2 -25739.794} C_VEL
LIN {X 0,Y 123.126,Z 216.15,A -85,B 0,C 180,E1 -25741.634,E2 -25741.634} C_VEL
LIN {X 0,Y 124.157,Z 218.575,A -85,B 0,C 180,E1 -25749.556,E2 -25749.556} C_VEL
LIN {X 0,Y 124.782,Z 220.286,A -85,B 0,C 180,E1 -25752.142,E2 -25752.142} C_VEL
LIN {X 0,Y 125.32,Z 222.966,A -85,B 0,C 180,E1 -25754.562,E2 -25754.562} C_VEL
LIN {X 0,Y 126.854,Z 231.242,A -85,B 0,C 180,E1 -25760.774,E2 -25760.774} C_VEL
LIN {X 0,Y 127.646,Z 232.835,A -85,B 0,C 180,E1 -25762.392,E2 -25762.392} C_VEL
LIN {X 0,Y 130.552,Z 237.589,A -85,B 0,C 180,E1 -25767.229,E2 -25767.229} C_VEL
LIN {X 0,Y 132.532,Z 241.036,A -85,B 0,C 180,E1 -25770.248,E2 -25770.248} C_VEL
LIN {X 0,Y 135.897,Z 248.719,A -85,B 0,C 180,E1 -25775.575,E2 -25775.575} C_VEL
LIN {X 0,Y 138.297,Z 255.006,A -85,B 0,C 180,E1 -25779.437,E2 -25779.437} C_VEL
LIN {X 0,Y 140.413,Z 262.223,A -85,B 0,C 180,E1 -25783.487,E2 -25783.487} C_VEL
LIN {X 0,Y 141.829,Z 269.575,A -85,B 0,C 180,E1 -25787.415,E2 -25787.415} C_VEL
LIN {X 0,Y 142.677,Z 278.08,A -85,B 0,C 180,E1 -25792.008,E2 -25792.008} C_VEL
LIN {X 0,Y 143.111,Z 285.863,A -85,B 0,C 180,E1 -25796.597,E2 -25796.597} C_VEL
LIN {X 0,Y 144.595,Z 292.102,A -85,B 0,C 180,E1 -25801.028,E2 -25801.028} C_VEL
LIN {X 0,Y 147.08,Z 297.072,A -85,B 0,C 180,E1 -25805.211,E2 -25805.211} C_VEL
LIN {X 0,Y 150.436,Z 301.063,A -85,B 0,C 180,E1 -25809.119,E2 -25809.119} C_VEL
LIN {X 0,Y 154.508,Z 304.297,A -85,B 0,C 180,E1 -25812.782,E2 -25812.782} C_VEL
LIN {X 0,Y 161.408,Z 307.603,A -85,B 0,C 180,E1 -25817.426,E2 -25817.426} C_VEL
LIN {X 0,Y 170.288,Z 310.044,A -85,B 0,C 180,E1 -25822.09,E2 -25822.09} C_VEL
LIN {X 0,Y 178.096,Z 311.227,A -85,B 0,C 180,E1 -25825.473,E2 -25825.473} C_VEL
LIN {X 0,Y 184.239,Z 311.616,A -85,B 0,C 180,E1 -25827.814,E2 -25827.814} C_VEL
LIN {X 0,Y 190.412,Z 311.588,A -85,B 0,C 180,E1 -25830,E2 -25830} C_VEL
LIN {X 0,Y 182.92,Z 311.538,A -85,B 0,C 180,E1 -25832.654,E2 -25832.654} C_VEL
LIN {X 0,Y 176.42,Z 311.068,A -85,B 0,C 180,E1 -25835.193,E2 -25835.193} C_VEL
LIN {X 0,Y 166.561,Z 309.195,A -85,B 0,C 180,E1 -25839.717,E2 -25839.717} C_VEL
LIN {X 0,Y 159.259,Z 306.707,A -85,B 0,C 180,E1 -25843.876,E2 -25843.876} C_VEL
LIN {X 0,Y 154.508,Z 304.297,A -85,B 0,C 180,E1 -25847.218,E2 -25847.218} C_VEL
LIN {X 0,Y 149.215,Z 299.883,A -85,B 0,C 180,E1 -25852.135,E2 -25852.135} C_VEL
LIN {X 0,Y 145.461,Z 294.162,A -85,B 0,C 180,E1 -25857.322,E2 -25857.322} C_VEL
LIN {X 0,Y 143.567,Z 288.309,A -85,B 0,C 180,E1 -25861.751,E2 -25861.751} C_VEL
LIN {X 0,Y 142.764,Z 282.792,A -85,B 0,C 180,E1 -25865.344,E2 -25865.344} C_VEL
LIN {X 0,Y 142.527,Z 275.908,A -85,B 0,C 180,E1 -25869.174,E2 -25869.174} C_VEL
LIN {X 0,Y 141.645,Z 268.573,A -85,B 0,C 180,E1 -25873.105,E2 -25873.105} C_VEL
LIN {X 0,Y 140.016,Z 260.687,A -85,B 0,C 180,E1 -25877.344,E2 -25877.344} C_VEL
LIN {X 0,Y 137.64,Z 253.078,A -85,B 0,C 180,E1 -25881.737,E2 -25881.737} C_VEL
LIN {X 0,Y 134.924,Z 246.463,A -85,B 0,C 180,E1 -25885.961,E2 -25885.961} C_VEL
LIN {X 0,Y 132.519,Z 241.07,A -85,B 0,C 180,E1 -25889.749,E2 -25889.749} C_VEL
LIN {X 0,Y 129.605,Z 236.099,A -85,B 0,C 180,E1 -25894.292,E2 -25894.292} C_VEL
LIN {X 0,Y 126.927,Z 231.749,A -85,B 0,C 180,E1 -25898.907,E2 -25898.907} C_VEL
LIN {X 0,Y 125.013,Z 228.936,A -85,B 0,C 180,E1 -25902.881,E2 -25902.881} C_VEL
LIN {X 0,Y 124.796,Z 228.183,A -85,B 0,C 180,E1 -25903.647,E2 -25903.647} C_VEL
LIN {X 0,Y 122.849,Z 226.014,A -85,B 0,C 180,E1 -25908.869,E2 -25908.869} C_VEL
LIN {X 0,Y 121.577,Z 222.598,A -85,B 0,C 180,E1 -25920.002,E2 -25920.002} C_VEL
LIN {X 0,Y 124.628,Z 227.628,A -85,B 0,C 180,E1 -25934.702,E2 -25934.702} C_VEL
LIN {X 0,Y 126.424,Z 232.138,A -85,B 0,C 180,E1 -25939.486,E2 -25939.486} C_VEL
LIN {X 0,Y 127.295,Z 233.321,A -85,B 0,C 180,E1 -25941.032,E2 -25941.032} C_VEL
LIN {X 0,Y 130.238,Z 239.127,A -85,B 0,C 180,E1 -25946.138,E2 -25946.138} C_VEL
LIN {X 0,Y 132.949,Z 246.344,A -85,B 0,C 180,E1 -25951.027,E2 -25951.027} C_VEL
LIN {X 0,Y 134.634,Z 251.266,A -85,B 0,C 180,E1 -25953.986,E2 -25953.986} C_VEL
LIN {X 0,Y 136.061,Z 256.928,A -85,B 0,C 180,E1 -25956.983,E2 -25956.983} C_VEL
LIN {X 0,Y 136.609,Z 262.343,A -85,B 0,C 180,E1 -25959.495,E2 -25959.495} C_VEL
LIN {X 0,Y 136.388,Z 269.725,A -85,B 0,C 180,E1 -25962.584,E2 -25962.584} C_VEL
LIN {X 0,Y 135.409,Z 278.002,A -85,B 0,C 180,E1 -25966.156,E2 -25966.156} C_VEL
LIN {X 0,Y 134.099,Z 284.42,A -85,B 0,C 180,E1 -25969.073,E2 -25969.073} C_VEL
LIN {X 0,Y 132.499,Z 289.351,A -85,B 0,C 180,E1 -25971.447,E2 -25971.447} C_VEL
LIN {X 0,Y 127.346,Z 297.685,A -85,B 0,C 180,E1 -25975.551,E2 -25975.551} C_VEL
LIN {X 0,Y 123.653,Z 303.35,A -85,B 0,C 180,E1 -25979.235,E2 -25979.235} C_VEL
LIN {X 0,Y 119.645,Z 308.843,A -85,B 0,C 180,E1 -25983.861,E2 -25983.861} C_VEL
LIN {X 0,Y 116.422,Z 313.171,A -85,B 0,C 180,E1 -25988.765,E2 -25988.765} C_VEL
LIN {X 0,Y 114.855,Z 315.546,A -85,B 0,C 180,E1 -25992.185,E2 -25992.185} C_VEL
LIN {X 0,Y 113.66,Z 317.353,A -85,B 0,C 180,E1 -25995.68,E2 -25995.68} C_VEL
LIN {X 0,Y 112.342,Z 319.816,A -85,B 0,C 180,E1 -26002.813,E2 -26002.813} C_VEL
LIN {X 0,Y 112.14,Z 320.413,A -85,B 0,C 180,E1 -26006.407,E2 -26006.407} C_VEL
LIN {X 0,Y 112.265,Z 320.576,A -85,B 0,C 180,E1 -26010,E2 -26010} C_VEL
LIN {X 0,Y 112.14,Z 320.413,A -85,B 0,C 180,E1 -26013.593,E2 -26013.593} C_VEL
LIN {X 0,Y 112.342,Z 319.816,A -85,B 0,C 180,E1 -26017.187,E2 -26017.187} C_VEL
LIN {X 0,Y 113.66,Z 317.353,A -85,B 0,C 180,E1 -26024.32,E2 -26024.32} C_VEL
LIN {X 0,Y 115.573,Z 314.391,A -85,B 0,C 180,E1 -26029.539,E2 -26029.539} C_VEL
LIN {X 0,Y 118.483,Z 310.398,A -85,B 0,C 180,E1 -26034.532,E2 -26034.532} C_VEL
LIN {X 0,Y 122.203,Z 305.265,A -85,B 0,C 180,E1 -26039.264,E2 -26039.264} C_VEL
LIN {X 0,Y 126.103,Z 299.556,A -85,B 0,C 180,E1 -26043.279,E2 -26043.279} C_VEL
LIN {X 0,Y 129.831,Z 293.677,A -85,B 0,C 180,E1 -26046.544,E2 -26046.544} C_VEL
LIN {X 0,Y 132.492,Z 289.351,A -85,B 0,C 180,E1 -26048.555,E2 -26048.555} C_VEL
LIN {X 0,Y 133.591,Z 286.066,A -85,B 0,C 180,E1 -26050.124,E2 -26050.124} C_VEL
LIN {X 0,Y 134.908,Z 280.701,A -85,B 0,C 180,E1 -26052.627,E2 -26052.627} C_VEL
LIN {X 0,Y 136.029,Z 273.548,A -85,B 0,C 180,E1 -26055.794,E2 -26055.794} C_VEL
LIN {X 0,Y 136.582,Z 265.33,A -85,B 0,C 180,E1 -26059.279,E2 -26059.279} C_VEL
LIN {X 0,Y 136.426,Z 259.483,A -85,B 0,C 180,E1 -26061.815,E2 -26061.815} C_VEL
LIN {X 0,Y 135.593,Z 254.841,A -85,B 0,C 180,E1 -26064.057,E2 -26064.057} C_VEL
LIN {X 0,Y 133.457,Z 247.49,A -85,B 0,C 180,E1 -26068.221,E2 -26068.221} C_VEL
LIN {X 0,Y 131.581,Z 242.865,A -85,B 0,C 180,E1 -26071.267,E2 -26071.267} C_VEL
LIN {X 0,Y 129.908,Z 238.599,A -85,B 0,C 180,E1 -26074.353,E2 -26074.353} C_VEL
LIN {X 0,Y 127.307,Z 233.285,A -85,B 0,C 180,E1 -26078.97,E2 -26078.97} C_VEL
LIN {X 0,Y 125.842,Z 231.207,A -85,B 0,C 180,E1 -26081.695,E2 -26081.695} C_VEL
LIN {X 0,Y 124.635,Z 227.6,A -85,B 0,C 180,E1 -26085.299,E2 -26085.299} C_VEL
LIN {X 0,Y 121.573,Z 222.612,A -85,B 0,C 180,E1 -26099.998,E2 -26099.998} C_VEL
LIN {X 0,Y 123.553,Z 226.683,A -85,B 0,C 180,E1 -26113.15,E2 -26113.15} C_VEL
LIN {X 0,Y 124.794,Z 228.19,A -85,B 0,C 180,E1 -26116.353,E2 -26116.353} C_VEL
LIN {X 0,Y 126.048,Z 230.789,A -85,B 0,C 180,E1 -26119.543,E2 -26119.543} C_VEL
LIN {X 0,Y 127.646,Z 232.835,A -85,B 0,C 180,E1 -26122.392,E2 -26122.392} C_VEL
LIN {X 0,Y 128.789,Z 235.544,A -85,B 0,C 180,E1 -26124.678,E2 -26124.678} C_VEL
LIN {X 0,Y 129.304,Z 239.176,A -85,B 0,C 180,E1 -26126.764,E2 -26126.764} C_VEL
LIN {X 0,Y 129.975,Z 249.862,A -85,B 0,C 180,E1 -26132.11,E2 -26132.11} C_VEL
LIN {X 0,Y 130.606,Z 252.08,A -85,B 0,C 180,E1 -26133.565,E2 -26133.565} C_VEL
LIN {X 0,Y 132.942,Z 258.825,A -85,B 0,C 180,E1 -26138.23,E2 -26138.23} C_VEL
LIN {X 0,Y 134.616,Z 265.303,A -85,B 0,C 180,E1 -26142.26,E2 -26142.26} C_VEL
LIN {X 0,Y 135.575,Z 270.805,A -85,B 0,C 180,E1 -26145.458,E2 -26145.458} C_VEL
LIN {X 0,Y 136.267,Z 278.13,A -85,B 0,C 180,E1 -26149.752,E2 -26149.752} C_VEL
LIN {X 0,Y 136.309,Z 285.898,A -85,B 0,C 180,E1 -26154.547,E2 -26154.547} C_VEL
LIN {X 0,Y 137.226,Z 292.201,A -85,B 0,C 180,E1 -26159.194,E2 -26159.194} C_VEL
LIN {X 0,Y 138.775,Z 296.512,A -85,B 0,C 180,E1 -26162.885,E2 -26162.885} C_VEL
LIN {X 0,Y 142.243,Z 301.426,A -85,B 0,C 180,E1 -26167.957,E2 -26167.957} C_VEL
LIN {X 0,Y 147.068,Z 305.376,A -85,B 0,C 180,E1 -26172.886,E2 -26172.886} C_VEL
LIN {X 0,Y 152.132,Z 307.886,A -85,B 0,C 180,E1 -26176.645,E2 -26176.645} C_VEL
LIN {X 0,Y 157.141,Z 309.482,A -85,B 0,C 180,E1 -26179.707,E2 -26179.707} C_VEL
LIN {X 0,Y 169.184,Z 311.557,A -85,B 0,C 180,E1 -26185.521,E2 -26185.521} C_VEL
LIN {X 0,Y 175.788,Z 311.96,A -85,B 0,C 180,E1 -26188.148,E2 -26188.148} C_VEL
LIN {X 0,Y 180.88,Z 311.866,A -85,B 0,C 180,E1 -26190,E2 -26190} C_VEL
LIN {X 0,Y 174.537,Z 311.902,A -85,B 0,C 180,E1 -26192.308,E2 -26192.308} C_VEL
LIN {X 0,Y 168.396,Z 311.512,A -85,B 0,C 180,E1 -26194.788,E2 -26194.788} C_VEL
LIN {X 0,Y 157.117,Z 309.475,A -85,B 0,C 180,E1 -26200.307,E2 -26200.307} C_VEL
LIN {X 0,Y 149.85,Z 306.842,A -85,B 0,C 180,E1 -26204.947,E2 -26204.947} C_VEL
LIN {X 0,Y 145.694,Z 304.519,A -85,B 0,C 180,E1 -26208.353,E2 -26208.353} C_VEL
LIN {X 0,Y 141.031,Z 300.147,A -85,B 0,C 180,E1 -26213.494,E2 -26213.494} C_VEL
LIN {X 0,Y 138.129,Z 295.057,A -85,B 0,C 180,E1 -26218.425,E2 -26218.425} C_VEL
LIN {X 0,Y 136.482,Z 288.339,A -85,B 0,C 180,E1 -26223.757,E2 -26223.757} C_VEL
LIN {X 0,Y 136.245,Z 281.461,A -85,B 0,C 180,E1 -26228.242,E2 -26228.242} C_VEL
LIN {X 0,Y 136.161,Z 276.508,A -85,B 0,C 180,E1 -26231.207,E2 -26231.207} C_VEL
LIN {X 0,Y 135.338,Z 269.179,A -85,B 0,C 180,E1 -26235.494,E2 -26235.494} C_VEL
LIN {X 0,Y 133.835,Z 261.873,A -85,B 0,C 180,E1 -26239.885,E2 -26239.885} C_VEL
LIN {X 0,Y 131.445,Z 254.182,A -85,B 0,C 180,E1 -26244.93,E2 -26244.93} C_VEL
LIN {X 0,Y 128.514,Z 246.704,A -85,B 0,C 180,E1 -26250.518,E2 -26250.518} C_VEL
LIN {X 0,Y 125.901,Z 241.797,A -85,B 0,C 180,E1 -26255.252,E2 -26255.252} C_VEL
LIN {X 0,Y 124.406,Z 238.85,A -85,B 0,C 180,E1 -26258.459,E2 -26258.459} C_VEL
LIN {X 0,Y 122.393,Z 235.517,A -85,B 0,C 180,E1 -26263.317,E2 -26263.317} C_VEL
LIN {X 0,Y 121.284,Z 233.562,A -85,B 0,C 180,E1 -26266.6,E2 -26266.6} C_VEL
LIN {X 0,Y 119.646,Z 229.527,A -85,B 0,C 180,E1 -26280.002,E2 -26280.002} C_VEL
LIN {X 0,Y 121.739,Z 233.872,A -85,B 0,C 180,E1 -26293.353,E2 -26293.353} C_VEL
LIN {X 0,Y 124.742,Z 240.75,A -85,B 0,C 180,E1 -26301.484,E2 -26301.484} C_VEL
LIN {X 0,Y 126.568,Z 245.196,A -85,B 0,C 180,E1 -26305.491,E2 -26305.491} C_VEL
LIN {X 0,Y 128.397,Z 250.725,A -85,B 0,C 180,E1 -26309.515,E2 -26309.515} C_VEL
LIN {X 0,Y 130,Z 256.287,A -85,B 0,C 180,E1 -26313.135,E2 -26313.135} C_VEL
LIN {X 0,Y 131.016,Z 262.072,A -85,B 0,C 180,E1 -26316.426,E2 -26316.426} C_VEL
LIN {X 0,Y 131.06,Z 267.695,A -85,B 0,C 180,E1 -26319.057,E2 -26319.057} C_VEL
LIN {X 0,Y 130.215,Z 275.57,A -85,B 0,C 180,E1 -26322.664,E2 -26322.664} C_VEL
LIN {X 0,Y 128.384,Z 284.248,A -85,B 0,C 180,E1 -26326.858,E2 -26326.858} C_VEL
LIN {X 0,Y 126.869,Z 289.134,A -85,B 0,C 180,E1 -26329.391,E2 -26329.391} C_VEL
LIN {X 0,Y 122.39,Z 296.218,A -85,B 0,C 180,E1 -26332.92,E2 -26332.92} C_VEL
LIN {X 0,Y 117.558,Z 303.137,A -85,B 0,C 180,E1 -26337.45,E2 -26337.45} C_VEL
LIN {X 0,Y 113.278,Z 308.631,A -85,B 0,C 180,E1 -26342.27,E2 -26342.27} C_VEL
LIN {X 0,Y 109.814,Z 312.96,A -85,B 0,C 180,E1 -26347.419,E2 -26347.419} C_VEL
LIN {X 0,Y 108.068,Z 315.333,A -85,B 0,C 180,E1 -26351.025,E2 -26351.025} C_VEL
LIN {X 0,Y 106.766,Z 317.14,A -85,B 0,C 180,E1 -26354.734,E2 -26354.734} C_VEL
LIN {X 0,Y 105.285,Z 319.605,A -85,B 0,C 180,E1 -26362.328,E2 -26362.328} C_VEL
LIN {X 0,Y 105.049,Z 320.202,A -85,B 0,C 180,E1 -26366.164,E2 -26366.164} C_VEL
LIN {X 0,Y 105.177,Z 320.365,A -85,B 0,C 180,E1 -26370,E2 -26370} C_VEL
LIN {X 0,Y 105.049,Z 320.202,A -85,B 0,C 180,E1 -26373.836,E2 -26373.836} C_VEL
LIN {X 0,Y 105.285,Z 319.605,A -85,B 0,C 180,E1 -26377.672,E2 -26377.672} C_VEL
LIN {X 0,Y 106.766,Z 317.14,A -85,B 0,C 180,E1 -26385.266,E2 -26385.266} C_VEL
LIN {X 0,Y 108.879,Z 314.179,A -85,B 0,C 180,E1 -26390.794,E2 -26390.794} C_VEL
LIN {X 0,Y 112.047,Z 310.186,A -85,B 0,C 180,E1 -26396.044,E2 -26396.044} C_VEL
LIN {X 0,Y 116.053,Z 305.053,A -85,B 0,C 180,E1 -26400.98,E2 -26400.98} C_VEL
LIN {X 0,Y 119.733,Z 299.984,A -85,B 0,C 180,E1 -26404.735,E2 -26404.735} C_VEL
LIN {X 0,Y 124.169,Z 293.464,A -85,B 0,C 180,E1 -26408.506,E2 -26408.506} C_VEL
LIN {X 0,Y 126.856,Z 289.133,A -85,B 0,C 180,E1 -26410.614,E2 -26410.614} C_VEL
LIN {X 0,Y 128.929,Z 282.031,A -85,B 0,C 180,E1 -26414.241,E2 -26414.241} C_VEL
LIN {X 0,Y 130.377,Z 274.463,A -85,B 0,C 180,E1 -26417.831,E2 -26417.831} C_VEL
LIN {X 0,Y 131.142,Z 265.449,A -85,B 0,C 180,E1 -26421.954,E2 -26421.954} C_VEL
LIN {X 0,Y 130.729,Z 259.758,A -85,B 0,C 180,E1 -26424.84,E2 -26424.84} C_VEL
LIN {X 0,Y 129.148,Z 253.028,A -85,B 0,C 180,E1 -26428.869,E2 -26428.869} C_VEL
LIN {X 0,Y 127.7,Z 248.479,A -85,B 0,C 180,E1 -26432.105,E2 -26432.105} C_VEL
LIN {X 0,Y 126.179,Z 244.242,A -85,B 0,C 180,E1 -26435.306,E2 -26435.306} C_VEL
LIN {X 0,Y 125.328,Z 242.703,A -85,B 0,C 180,E1 -26436.886,E2 -26436.886} C_VEL
LIN {X 0,Y 124.751,Z 240.727,A -85,B 0,C 180,E1 -26438.518,E2 -26438.518} C_VEL
LIN {X 0,Y 123.522,Z 238.317,A -85,B 0,C 180,E1 -26441.338,E2 -26441.338} C_VEL
LIN {X 0,Y 121.738,Z 233.876,A -85,B 0,C 180,E1 -26446.647,E2 -26446.647} C_VEL
LIN {X 0,Y 119.635,Z 229.561,A -85,B 0,C 180,E1 -26459.998,E2 -26459.998} C_VEL
LIN {X 0,Y 121.278,Z 233.581,A -85,B 0,C 180,E1 -26473.401,E2 -26473.401} C_VEL
LIN {X 0,Y 123.664,Z 237.726,A -85,B 0,C 180,E1 -26479.935,E2 -26479.935} C_VEL
LIN {X 0,Y 124.405,Z 238.852,A -85,B 0,C 180,E1 -26481.541,E2 -26481.541} C_VEL
LIN {X 0,Y 126.8,Z 243.256,A -85,B 0,C 180,E1 -26486.32,E2 -26486.32} C_VEL
LIN {X 0,Y 128.868,Z 247.766,A -85,B 0,C 180,E1 -26490.294,E2 -26490.294} C_VEL
LIN {X 0,Y 130.606,Z 252.08,A -85,B 0,C 180,E1 -26493.565,E2 -26493.565} C_VEL
LIN {X 0,Y 131.23,Z 254.269,A -85,B 0,C 180,E1 -26494.971,E2 -26494.971} C_VEL
LIN {X 0,Y 131.41,Z 258.147,A -85,B 0,C 180,E1 -26496.927,E2 -26496.927} C_VEL
LIN {X 0,Y 130.945,Z 262.353,A -85,B 0,C 180,E1 -26498.766,E2 -26498.766} C_VEL
LIN {X 0,Y 129.482,Z 271.43,A -85,B 0,C 180,E1 -26502.952,E2 -26502.952} C_VEL
LIN {X 0,Y 129.499,Z 273.173,A -85,B 0,C 180,E1 -26504.032,E2 -26504.032} C_VEL
LIN {X 0,Y 129.954,Z 280.131,A -85,B 0,C 180,E1 -26508.513,E2 -26508.513} C_VEL
LIN {X 0,Y 129.792,Z 286.139,A -85,B 0,C 180,E1 -26512.471,E2 -26512.471} C_VEL
LIN {X 0,Y 130.139,Z 292.449,A -85,B 0,C 180,E1 -26517.314,E2 -26517.314} C_VEL
LIN {X 0,Y 131.971,Z 298.493,A -85,B 0,C 180,E1 -26522.996,E2 -26522.996} C_VEL
LIN {X 0,Y 134.272,Z 301.971,A -85,B 0,C 180,E1 -26526.886,E2 -26526.886} C_VEL
LIN {X 0,Y 138.933,Z 306.002,A -85,B 0,C 180,E1 -26532.332,E2 -26532.332} C_VEL
LIN {X 0,Y 144.383,Z 308.646,A -85,B 0,C 180,E1 -26536.778,E2 -26536.778} C_VEL
LIN {X 0,Y 149.753,Z 310.328,A -85,B 0,C 180,E1 -26540.235,E2 -26540.235} C_VEL
LIN {X 0,Y 158.821,Z 311.793,A -85,B 0,C 180,E1 -26544.923,E2 -26544.923} C_VEL
LIN {X 0,Y 168.692,Z 312.223,A -85,B 0,C 180,E1 -26549.034,E2 -26549.034} C_VEL
LIN {X 0,Y 171.243,Z 312.148,A -85,B 0,C 180,E1 -26550,E2 -26550} C_VEL
LIN {X 0,Y 161.969,Z 312.002,A -85,B 0,C 180,E1 -26553.654,E2 -26553.654} C_VEL
LIN {X 0,Y 153.03,Z 310.939,A -85,B 0,C 180,E1 -26557.919,E2 -26557.919} C_VEL
LIN {X 0,Y 147.759,Z 309.758,A -85,B 0,C 180,E1 -26560.968,E2 -26560.968} C_VEL
LIN {X 0,Y 143.036,Z 308.165,A -85,B 0,C 180,E1 -26564.221,E2 -26564.221} C_VEL
LIN {X 0,Y 137.316,Z 304.881,A -85,B 0,C 180,E1 -26569.403,E2 -26569.403} C_VEL
LIN {X 0,Y 132.626,Z 299.702,A -85,B 0,C 180,E1 -26575.734,E2 -26575.734} C_VEL
LIN {X 0,Y 130.622,Z 294.854,A -85,B 0,C 180,E1 -26580.59,E2 -26580.59} C_VEL
LIN {X 0,Y 129.731,Z 288.754,A -85,B 0,C 180,E1 -26585.652,E2 -26585.652} C_VEL
LIN {X 0,Y 129.924,Z 282.63,A -85,B 0,C 180,E1 -26589.879,E2 -26589.879} C_VEL
LIN {X 0,Y 129.813,Z 276.661,A -85,B 0,C 180,E1 -26593.768,E2 -26593.768} C_VEL
LIN {X 0,Y 129.027,Z 269.443,A -85,B 0,C 180,E1 -26598.428,E2 -26598.428} C_VEL
LIN {X 0,Y 127.723,Z 263.066,A -85,B 0,C 180,E1 -26602.753,E2 -26602.753} C_VEL
LIN {X 0,Y 125.633,Z 256.226,A -85,B 0,C 180,E1 -26607.898,E2 -26607.898} C_VEL
LIN {X 0,Y 124.094,Z 251.79,A -85,B 0,C 180,E1 -26611.638,E2 -26611.638} C_VEL
LIN {X 0,Y 122.069,Z 247.409,A -85,B 0,C 180,E1 -26616.235,E2 -26616.235} C_VEL
LIN {X 0,Y 120.834,Z 244.627,A -85,B 0,C 180,E1 -26619.577,E2 -26619.577} C_VEL
LIN {X 0,Y 118.627,Z 240.446,A -85,B 0,C 180,E1 -26626.294,E2 -26626.294} C_VEL
LIN {X 0,Y 117.243,Z 238.234,A -85,B 0,C 180,E1 -26633.116,E2 -26633.116} C_VEL
LIN {X 0,Y 117.319,Z 236.34,A -85,B 0,C 180,E1 -26640.002,E2 -26640.002} C_VEL
LIN {X 0,Y 118.201,Z 239.492,A -85,B 0,C 180,E1 -26650.277,E2 -26650.277} C_VEL
LIN {X 0,Y 119.131,Z 240.934,A -85,B 0,C 180,E1 -26653.651,E2 -26653.651} C_VEL
LIN {X 0,Y 121.135,Z 246.41,A -85,B 0,C 180,E1 -26660.374,E2 -26660.374} C_VEL
LIN {X 0,Y 122.612,Z 250.753,A -85,B 0,C 180,E1 -26664.557,E2 -26664.557} C_VEL
LIN {X 0,Y 124.687,Z 258.52,A -85,B 0,C 180,E1 -26670.485,E2 -26670.485} C_VEL
LIN {X 0,Y 125.682,Z 265.028,A -85,B 0,C 180,E1 -26674.666,E2 -26674.666} C_VEL
LIN {X 0,Y 125.51,Z 270.139,A -85,B 0,C 180,E1 -26677.384,E2 -26677.384} C_VEL
LIN {X 0,Y 124.557,Z 276.575,A -85,B 0,C 180,E1 -26680.544,E2 -26680.544} C_VEL
LIN {X 0,Y 122.663,Z 284.608,A -85,B 0,C 180,E1 -26684.719,E2 -26684.719} C_VEL
LIN {X 0,Y 120.614,Z 290.49,A -85,B 0,C 180,E1 -26687.927,E2 -26687.927} C_VEL
LIN {X 0,Y 114.951,Z 298.417,A -85,B 0,C 180,E1 -26692.31,E2 -26692.31} C_VEL
LIN {X 0,Y 111.585,Z 302.924,A -85,B 0,C 180,E1 -26695.47,E2 -26695.47} C_VEL
LIN {X 0,Y 107,Z 308.418,A -85,B 0,C 180,E1 -26700.488,E2 -26700.488} C_VEL
LIN {X 0,Y 103.281,Z 312.748,A -85,B 0,C 180,E1 -26705.903,E2 -26705.903} C_VEL
LIN {X 0,Y 101.336,Z 315.12,A -85,B 0,C 180,E1 -26709.711,E2 -26709.711} C_VEL
LIN {X 0,Y 99.891,Z 316.928,A -85,B 0,C 180,E1 -26713.655,E2 -26713.655} C_VEL
LIN {X 0,Y 98.253,Z 319.393,A -85,B 0,C 180,E1 -26721.775,E2 -26721.775} C_VEL
LIN {X 0,Y 97.955,Z 319.99,A -85,B 0,C 180,E1 -26725.886,E2 -26725.886} C_VEL
LIN {X 0,Y 98.081,Z 320.154,A -85,B 0,C 180,E1 -26730,E2 -26730} C_VEL
LIN {X 0,Y 97.955,Z 319.99,A -85,B 0,C 180,E1 -26734.114,E2 -26734.114} C_VEL
LIN {X 0,Y 98.253,Z 319.393,A -85,B 0,C 180,E1 -26738.225,E2 -26738.225} C_VEL
LIN {X 0,Y 99.891,Z 316.928,A -85,B 0,C 180,E1 -26746.345,E2 -26746.345} C_VEL
LIN {X 0,Y 102.252,Z 313.967,A -85,B 0,C 180,E1 -26752.211,E2 -26752.211} C_VEL
LIN {X 0,Y 105.697,Z 309.974,A -85,B 0,C 180,E1 -26757.738,E2 -26757.738} C_VEL
LIN {X 0,Y 110.012,Z 304.842,A -85,B 0,C 180,E1 -26762.888,E2 -26762.888} C_VEL
LIN {X 0,Y 113.481,Z 300.375,A -85,B 0,C 180,E1 -26766.377,E2 -26766.377} C_VEL
LIN {X 0,Y 117.709,Z 294.629,A -85,B 0,C 180,E1 -26769.929,E2 -26769.929} C_VEL
LIN {X 0,Y 120.597,Z 290.489,A -85,B 0,C 180,E1 -26772.08,E2 -26772.08} C_VEL
LIN {X 0,Y 123.091,Z 283.133,A -85,B 0,C 180,E1 -26776.109,E2 -26776.109} C_VEL
LIN {X 0,Y 125.023,Z 274.191,A -85,B 0,C 180,E1 -26780.631,E2 -26780.631} C_VEL
LIN {X 0,Y 125.756,Z 267.458,A -85,B 0,C 180,E1 -26784.012,E2 -26784.012} C_VEL
LIN {X 0,Y 125.326,Z 262.364,A -85,B 0,C 180,E1 -26786.948,E2 -26786.948} C_VEL
LIN {X 0,Y 124.375,Z 257.163,A -85,B 0,C 180,E1 -26790.479,E2 -26790.479} C_VEL
LIN {X 0,Y 122.329,Z 249.817,A -85,B 0,C 180,E1 -26796.285,E2 -26796.285} C_VEL
LIN {X 0,Y 120.533,Z 244.912,A -85,B 0,C 180,E1 -26801.293,E2 -26801.293} C_VEL
LIN {X 0,Y 119.133,Z 240.931,A -85,B 0,C 180,E1 -26806.349,E2 -26806.349} C_VEL
LIN {X 0,Y 118.202,Z 239.489,A -85,B 0,C 180,E1 -26809.723,E2 -26809.723} C_VEL
LIN {X 0,Y 117.312,Z 236.36,A -85,B 0,C 180,E1 -26819.998,E2 -26819.998} C_VEL
LIN {X 0,Y 117.786,Z 239.198,A -85,B 0,C 180,E1 -26830.31,E2 -26830.31} C_VEL
LIN {X 0,Y 118.622,Z 240.457,A -85,B 0,C 180,E1 -26833.707,E2 -26833.707} C_VEL
LIN {X 0,Y 120.838,Z 244.617,A -85,B 0,C 180,E1 -26840.422,E2 -26840.422} C_VEL
LIN {X 0,Y 122.799,Z 248.798,A -85,B 0,C 180,E1 -26845.417,E2 -26845.417} C_VEL
LIN {X 0,Y 124.539,Z 252.996,A -85,B 0,C 180,E1 -26849.388,E2 -26849.388} C_VEL
LIN {X 0,Y 126.661,Z 259.508,A -85,B 0,C 180,E1 -26854.66,E2 -26854.66} C_VEL
LIN {X 0,Y 128.165,Z 265.173,A -85,B 0,C 180,E1 -26858.739,E2 -26858.739} C_VEL
LIN {X 0,Y 129.346,Z 271.625,A -85,B 0,C 180,E1 -26863.016,E2 -26863.016} C_VEL
LIN {X 0,Y 129.499,Z 273.173,A -85,B 0,C 180,E1 -26864.032,E2 -26864.032} C_VEL
LIN {X 0,Y 129.375,Z 275.629,A -85,B 0,C 180,E1 -26865.429,E2 -26865.429} C_VEL
LIN {X 0,Y 128.728,Z 278.272,A -85,B 0,C 180,E1 -26866.74,E2 -26866.74} C_VEL
LIN {X 0,Y 126.541,Z 283.431,A -85,B 0,C 180,E1 -26869.276,E2 -26869.276} C_VEL
LIN {X 0,Y 123.808,Z 289.471,A -85,B 0,C 180,E1 -26872.698,E2 -26872.698} C_VEL
LIN {X 0,Y 123.238,Z 292.494,A -85,B 0,C 180,E1 -26875.051,E2 -26875.051} C_VEL
LIN {X 0,Y 123.884,Z 297.018,A -85,B 0,C 180,E1 -26879.298,E2 -26879.298} C_VEL
LIN {X 0,Y 126.307,Z 302.362,A -85,B 0,C 180,E1 -26885.49,E2 -26885.49} C_VEL
LIN {X 0,Y 130.419,Z 306.269,A -85,B 0,C 180,E1 -26891.136,E2 -26891.136} C_VEL
LIN {X 0,Y 134.079,Z 308.44,A -85,B 0,C 180,E1 -26894.806,E2 -26894.806} C_VEL
LIN {X 0,Y 142.374,Z 311,A -85,B 0,C 180,E1 -26900.834,E2 -26900.834} C_VEL
LIN {X 0,Y 149.169,Z 312.079,A -85,B 0,C 180,E1 -26904.593,E2 -26904.593} C_VEL
LIN {X 0,Y 155.241,Z 312.467,A -85,B 0,C 180,E1 -26907.405,E2 -26907.405} C_VEL
LIN {X 0,Y 161.587,Z 312.43,A -85,B 0,C 180,E1 -26910,E2 -26910} C_VEL
LIN {X 0,Y 154.794,Z 312.441,A -85,B 0,C 180,E1 -26912.78,E2 -26912.78} C_VEL
LIN {X 0,Y 148.349,Z 312.019,A -85,B 0,C 180,E1 -26915.822,E2 -26915.822} C_VEL
LIN {X 0,Y 138.495,Z 310.039,A -85,B 0,C 180,E1 -26921.711,E2 -26921.711} C_VEL
LIN {X 0,Y 132.216,Z 307.452,A -85,B 0,C 180,E1 -26926.91,E2 -26926.91} C_VEL
LIN {X 0,Y 127.394,Z 303.693,A -85,B 0,C 180,E1 -26932.716,E2 -26932.716} C_VEL
LIN {X 0,Y 125.279,Z 300.665,A -85,B 0,C 180,E1 -26936.666,E2 -26936.666} C_VEL
LIN {X 0,Y 123.444,Z 294.809,A -85,B 0,C 180,E1 -26942.837,E2 -26942.837} C_VEL
LIN {X 0,Y 123.238,Z 288.923,A -85,B 0,C 180,E1 -26947.905,E2 -26947.905} C_VEL
LIN {X 0,Y 123.676,Z 282.825,A -85,B 0,C 180,E1 -26952.379,E2 -26952.379} C_VEL
LIN {X 0,Y 123.556,Z 276.393,A -85,B 0,C 180,E1 -26956.957,E2 -26956.957} C_VEL
LIN {X 0,Y 122.997,Z 270.741,A -85,B 0,C 180,E1 -26961.06,E2 -26961.06} C_VEL
LIN {X 0,Y 121.845,Z 265.105,A -85,B 0,C 180,E1 -26965.384,E2 -26965.384} C_VEL
LIN {X 0,Y 120.348,Z 259.42,A -85,B 0,C 180,E1 -26970.244,E2 -26970.244} C_VEL
LIN {X 0,Y 118.658,Z 254.306,A -85,B 0,C 180,E1 -26975.508,E2 -26975.508} C_VEL
LIN {X 0,Y 116.94,Z 250.226,A -85,B 0,C 180,E1 -26980.7,E2 -26980.7} C_VEL
LIN {X 0,Y 115.492,Z 246.738,A -85,B 0,C 180,E1 -26986.813,E2 -26986.813} C_VEL
LIN {X 0,Y 114.235,Z 243.887,A -85,B 0,C 180,E1 -26996.475,E2 -26996.475} C_VEL
LIN {X 0,Y 114.511,Z 242.969,A -85,B 0,C 180,E1 -27000.002,E2 -27000.002} C_VEL
LIN {X 0,Y 115.34,Z 246.151,A -85,B 0,C 180,E1 -27010.535,E2 -27010.535} C_VEL
LIN {X 0,Y 116.147,Z 248.387,A -85,B 0,C 180,E1 -27014.502,E2 -27014.502} C_VEL
LIN {X 0,Y 117.251,Z 251.921,A -85,B 0,C 180,E1 -27019.251,E2 -27019.251} C_VEL
LIN {X 0,Y 118.409,Z 255.984,A -85,B 0,C 180,E1 -27023.438,E2 -27023.438} C_VEL
LIN {X 0,Y 119.687,Z 262.581,A -85,B 0,C 180,E1 -27028.978,E2 -27028.978} C_VEL
LIN {X 0,Y 120.352,Z 268.028,A -85,B 0,C 180,E1 -27032.844,E2 -27032.844} C_VEL
LIN {X 0,Y 120.209,Z 271.648,A -85,B 0,C 180,E1 -27035.066,E2 -27035.066} C_VEL
LIN {X 0,Y 119.25,Z 277.041,A -85,B 0,C 180,E1 -27037.965,E2 -27037.965} C_VEL
LIN {X 0,Y 117.353,Z 284.127,A -85,B 0,C 180,E1 -27041.845,E2 -27041.845} C_VEL
LIN {X 0,Y 115.154,Z 290.266,A -85,B 0,C 180,E1 -27045.424,E2 -27045.424} C_VEL
LIN {X 0,Y 113.38,Z 293.041,A -85,B 0,C 180,E1 -27047.013,E2 -27047.013} C_VEL
LIN {X 0,Y 108.32,Z 299.52,A -85,B 0,C 180,E1 -27050.924,E2 -27050.924} C_VEL
LIN {X 0,Y 104.095,Z 304.629,A -85,B 0,C 180,E1 -27054.98,E2 -27054.98} C_VEL
LIN {X 0,Y 99.433,Z 309.762,A -85,B 0,C 180,E1 -27060.346,E2 -27060.346} C_VEL
LIN {X 0,Y 95.702,Z 313.755,A -85,B 0,C 180,E1 -27066.178,E2 -27066.178} C_VEL
LIN {X 0,Y 93.062,Z 316.715,A -85,B 0,C 180,E1 -27072.418,E2 -27072.418} C_VEL
LIN {X 0,Y 91.2,Z 319.181,A -85,B 0,C 180,E1 -27081.134,E2 -27081.134} C_VEL
LIN {X 0,Y 90.885,Z 319.779,A -85,B 0,C 180,E1 -27085.565,E2 -27085.565} C_VEL
LIN {X 0,Y 90.978,Z 319.942,A -85,B 0,C 180,E1 -27090,E2 -27090} C_VEL
LIN {X 0,Y 90.885,Z 319.779,A -85,B 0,C 180,E1 -27094.435,E2 -27094.435} C_VEL
LIN {X 0,Y 91.2,Z 319.181,A -85,B 0,C 180,E1 -27098.866,E2 -27098.866} C_VEL
LIN {X 0,Y 93.062,Z 316.715,A -85,B 0,C 180,E1 -27107.582,E2 -27107.582} C_VEL
LIN {X 0,Y 95.702,Z 313.755,A -85,B 0,C 180,E1 -27113.822,E2 -27113.822} C_VEL
LIN {X 0,Y 99.433,Z 309.762,A -85,B 0,C 180,E1 -27119.654,E2 -27119.654} C_VEL
LIN {X 0,Y 104.102,Z 304.63,A -85,B 0,C 180,E1 -27125.018,E2 -27125.018} C_VEL
LIN {X 0,Y 109.37,Z 298.203,A -85,B 0,C 180,E1 -27129.984,E2 -27129.984} C_VEL
LIN {X 0,Y 114.377,Z 291.662,A -85,B 0,C 180,E1 -27133.73,E2 -27133.73} C_VEL
LIN {X 0,Y 116.366,Z 287.033,A -85,B 0,C 180,E1 -27136.447,E2 -27136.447} C_VEL
LIN {X 0,Y 118.515,Z 279.993,A -85,B 0,C 180,E1 -27140.434,E2 -27140.434} C_VEL
LIN {X 0,Y 119.98,Z 273.167,A -85,B 0,C 180,E1 -27144.141,E2 -27144.141} C_VEL
LIN {X 0,Y 120.383,Z 267.987,A -85,B 0,C 180,E1 -27147.161,E2 -27147.161} C_VEL
LIN {X 0,Y 119.501,Z 261.387,A -85,B 0,C 180,E1 -27151.932,E2 -27151.932} C_VEL
LIN {X 0,Y 118.064,Z 254.921,A -85,B 0,C 180,E1 -27157.627,E2 -27157.627} C_VEL
LIN {X 0,Y 117.272,Z 251.879,A -85,B 0,C 180,E1 -27160.753,E2 -27160.753} C_VEL
LIN {X 0,Y 116.08,Z 248.016,A -85,B 0,C 180,E1 -27165.983,E2 -27165.983} C_VEL
LIN {X 0,Y 115.346,Z 246.137,A -85,B 0,C 180,E1 -27169.466,E2 -27169.466} C_VEL
LIN {X 0,Y 114.507,Z 242.979,A -85,B 0,C 180,E1 -27179.998,E2 -27179.998} C_VEL
LIN {X 0,Y 114.933,Z 245.818,A -85,B 0,C 180,E1 -27190.569,E2 -27190.569} C_VEL
LIN {X 0,Y 115.636,Z 247.203,A -85,B 0,C 180,E1 -27194.068,E2 -27194.068} C_VEL
LIN {X 0,Y 116.946,Z 250.214,A -85,B 0,C 180,E1 -27199.299,E2 -27199.299} C_VEL
LIN {X 0,Y 118.675,Z 254.274,A -85,B 0,C 180,E1 -27204.488,E2 -27204.488} C_VEL
LIN {X 0,Y 119.95,Z 258.054,A -85,B 0,C 180,E1 -27208.496,E2 -27208.496} C_VEL
LIN {X 0,Y 121.533,Z 263.74,A -85,B 0,C 180,E1 -27213.464,E2 -27213.464} C_VEL
LIN {X 0,Y 122.67,Z 269.096,A -85,B 0,C 180,E1 -27217.713,E2 -27217.713} C_VEL
LIN {X 0,Y 123.413,Z 274.607,A -85,B 0,C 180,E1 -27221.803,E2 -27221.803} C_VEL
LIN {X 0,Y 123.666,Z 280.435,A -85,B 0,C 180,E1 -27225.917,E2 -27225.917} C_VEL
LIN {X 0,Y 123.564,Z 285.433,A -85,B 0,C 180,E1 -27229.46,E2 -27229.46} C_VEL
LIN {X 0,Y 123.238,Z 292.494,A -85,B 0,C 180,E1 -27235.051,E2 -27235.051} C_VEL
LIN {X 0,Y 122.863,Z 295.422,A -85,B 0,C 180,E1 -27237.474,E2 -27237.474} C_VEL
LIN {X 0,Y 121.091,Z 299.999,A -85,B 0,C 180,E1 -27241.513,E2 -27241.513} C_VEL
LIN {X 0,Y 120.132,Z 303.993,A -85,B 0,C 180,E1 -27245.755,E2 -27245.755} C_VEL
LIN {X 0,Y 121.023,Z 305.753,A -85,B 0,C 180,E1 -27248.369,E2 -27248.369} C_VEL
LIN {X 0,Y 125.306,Z 308.711,A -85,B 0,C 180,E1 -27253.714,E2 -27253.714} C_VEL
LIN {X 0,Y 129.534,Z 310.371,A -85,B 0,C 180,E1 -27257.574,E2 -27257.574} C_VEL
LIN {X 0,Y 139.623,Z 312.365,A -85,B 0,C 180,E1 -27264.222,E2 -27264.222} C_VEL
LIN {X 0,Y 147.658,Z 312.836,A -85,B 0,C 180,E1 -27268.179,E2 -27268.179} C_VEL
LIN {X 0,Y 151.909,Z 312.713,A -85,B 0,C 180,E1 -27270,E2 -27270} C_VEL
LIN {X 0,Y 145.552,Z 312.755,A -85,B 0,C 180,E1 -27272.768,E2 -27272.768} C_VEL
LIN {X 0,Y 139.622,Z 312.365,A -85,B 0,C 180,E1 -27275.778,E2 -27275.778} C_VEL
LIN {X 0,Y 129.381,Z 310.316,A -85,B 0,C 180,E1 -27282.549,E2 -27282.549} C_VEL
LIN {X 0,Y 124.807,Z 308.459,A -85,B 0,C 180,E1 -27286.813,E2 -27286.813} C_VEL
LIN {X 0,Y 120.964,Z 305.761,A -85,B 0,C 180,E1 -27291.633,E2 -27291.633} C_VEL
LIN {X 0,Y 117.678,Z 300.92,A -85,B 0,C 180,E1 -27298.54,E2 -27298.54} C_VEL
LIN {X 0,Y 116.515,Z 295.167,A -85,B 0,C 180,E1 -27304.961,E2 -27304.961} C_VEL
LIN {X 0,Y 116.965,Z 289.086,A -85,B 0,C 180,E1 -27310.404,E2 -27310.404} C_VEL
LIN {X 0,Y 117.504,Z 283.363,A -85,B 0,C 180,E1 -27314.97,E2 -27314.97} C_VEL
LIN {X 0,Y 117.471,Z 276.981,A -85,B 0,C 180,E1 -27320.011,E2 -27320.011} C_VEL
LIN {X 0,Y 117.004,Z 271.918,A -85,B 0,C 180,E1 -27324.154,E2 -27324.154} C_VEL
LIN {X 0,Y 115.987,Z 266.488,A -85,B 0,C 180,E1 -27329,E2 -27329} C_VEL
LIN {X 0,Y 115.203,Z 262.744,A -85,B 0,C 180,E1 -27332.774,E2 -27332.774} C_VEL
LIN {X 0,Y 113.721,Z 258.198,A -85,B 0,C 180,E1 -27338.237,E2 -27338.237} C_VEL
LIN {X 0,Y 112.966,Z 255.727,A -85,B 0,C 180,E1 -27341.878,E2 -27341.878} C_VEL
LIN {X 0,Y 112.212,Z 253.753,A -85,B 0,C 180,E1 -27345.493,E2 -27345.493} C_VEL
LIN {X 0,Y 111.595,Z 252.198,A -85,B 0,C 180,E1 -27349.112,E2 -27349.112} C_VEL
LIN {X 0,Y 111.404,Z 249.455,A -85,B 0,C 180,E1 -27360.002,E2 -27360.002} C_VEL
LIN {X 0,Y 111.994,Z 252.702,A -85,B 0,C 180,E1 -27370.853,E2 -27370.853} C_VEL
LIN {X 0,Y 112.558,Z 254.767,A -85,B 0,C 180,E1 -27374.465,E2 -27374.465} C_VEL
LIN {X 0,Y 113.253,Z 257.346,A -85,B 0,C 180,E1 -27378.078,E2 -27378.078} C_VEL
LIN {X 0,Y 113.97,Z 261.046,A -85,B 0,C 180,E1 -27382.337,E2 -27382.337} C_VEL
LIN {X 0,Y 114.834,Z 267.441,A -85,B 0,C 180,E1 -27388.086,E2 -27388.086} C_VEL
LIN {X 0,Y 114.982,Z 272.923,A -85,B 0,C 180,E1 -27392.269,E2 -27392.269} C_VEL
LIN {X 0,Y 114.501,Z 275.891,A -85,B 0,C 180,E1 -27394.094,E2 -27394.094} C_VEL
LIN {X 0,Y 112.281,Z 283.76,A -85,B 0,C 180,E1 -27398.753,E2 -27398.753} C_VEL
LIN {X 0,Y 109.15,Z 291.442,A -85,B 0,C 180,E1 -27403.584,E2 -27403.584} C_VEL
LIN {X 0,Y 107.172,Z 294.205,A -85,B 0,C 180,E1 -27405.176,E2 -27405.176} C_VEL
LIN {X 0,Y 101.34,Z 301.125,A -85,B 0,C 180,E1 -27409.72,E2 -27409.72} C_VEL
LIN {X 0,Y 96.546,Z 306.333,A -85,B 0,C 180,E1 -27414.384,E2 -27414.384} C_VEL
LIN {X 0,Y 91.83,Z 311.082,A -85,B 0,C 180,E1 -27420.168,E2 -27420.168} C_VEL
LIN {X 0,Y 88.084,Z 314.695,A -85,B 0,C 180,E1 -27426.489,E2 -27426.489} C_VEL
LIN {X 0,Y 86.292,Z 316.503,A -85,B 0,C 180,E1 -27430.988,E2 -27430.988} C_VEL
LIN {X 0,Y 84.177,Z 318.969,A -85,B 0,C 180,E1 -27440.388,E2 -27440.388} C_VEL
LIN {X 0,Y 83.801,Z 319.568,A -85,B 0,C 180,E1 -27445.189,E2 -27445.189} C_VEL
LIN {X 0,Y 83.885,Z 319.731,A -85,B 0,C 180,E1 -27450,E2 -27450} C_VEL
LIN {X 0,Y 83.801,Z 319.568,A -85,B 0,C 180,E1 -27454.811,E2 -27454.811} C_VEL
LIN {X 0,Y 84.177,Z 318.969,A -85,B 0,C 180,E1 -27459.612,E2 -27459.612} C_VEL
LIN {X 0,Y 86.292,Z 316.503,A -85,B 0,C 180,E1 -27469.012,E2 -27469.012} C_VEL
LIN {X 0,Y 89.217,Z 313.543,A -85,B 0,C 180,E1 -27475.674,E2 -27475.674} C_VEL
LIN {X 0,Y 93.285,Z 309.549,A -85,B 0,C 180,E1 -27481.827,E2 -27481.827} C_VEL
LIN {X 0,Y 98.331,Z 304.417,A -85,B 0,C 180,E1 -27487.41,E2 -27487.41} C_VEL
LIN {X 0,Y 104.005,Z 297.991,A -85,B 0,C 180,E1 -27492.511,E2 -27492.511} C_VEL
LIN {X 0,Y 108.243,Z 292.827,A -85,B 0,C 180,E1 -27495.577,E2 -27495.577} C_VEL
LIN {X 0,Y 110.507,Z 288.453,A -85,B 0,C 180,E1 -27498.354,E2 -27498.354} C_VEL
LIN {X 0,Y 113.089,Z 281.217,A -85,B 0,C 180,E1 -27502.772,E2 -27502.772} C_VEL
LIN {X 0,Y 114.775,Z 274.806,A -85,B 0,C 180,E1 -27506.555,E2 -27506.555} C_VEL
LIN {X 0,Y 114.982,Z 270.16,A -85,B 0,C 180,E1 -27509.715,E2 -27509.715} C_VEL
LIN {X 0,Y 114.695,Z 265.909,A -85,B 0,C 180,E1 -27513.227,E2 -27513.227} C_VEL
LIN {X 0,Y 113.84,Z 260.518,A -85,B 0,C 180,E1 -27518.257,E2 -27518.257} C_VEL
LIN {X 0,Y 113.284,Z 257.294,A -85,B 0,C 180,E1 -27521.927,E2 -27521.927} C_VEL
LIN {X 0,Y 112.295,Z 253.594,A -85,B 0,C 180,E1 -27527.345,E2 -27527.345} C_VEL
LIN {X 0,Y 112.01,Z 252.673,A -85,B 0,C 180,E1 -27529.148,E2 -27529.148} C_VEL
LIN {X 0,Y 111.4,Z 249.463,A -85,B 0,C 180,E1 -27539.998,E2 -27539.998} C_VEL
LIN {X 0,Y 111.595,Z 252.198,A -85,B 0,C 180,E1 -27550.888,E2 -27550.888} C_VEL
LIN {X 0,Y 112.199,Z 253.778,A -85,B 0,C 180,E1 -27554.508,E2 -27554.508} C_VEL
LIN {X 0,Y 113.308,Z 256.928,A -85,B 0,C 180,E1 -27559.944,E2 -27559.944} C_VEL
LIN {X 0,Y 114.704,Z 261.052,A -85,B 0,C 180,E1 -27565.395,E2 -27565.395} C_VEL
LIN {X 0,Y 115.594,Z 264.557,A -85,B 0,C 180,E1 -27569.101,E2 -27569.101} C_VEL
LIN {X 0,Y 116.612,Z 269.69,A -85,B 0,C 180,E1 -27573.88,E2 -27573.88} C_VEL
LIN {X 0,Y 117.259,Z 274.337,A -85,B 0,C 180,E1 -27577.902,E2 -27577.902} C_VEL
LIN {X 0,Y 117.563,Z 279.517,A -85,B 0,C 180,E1 -27582.007,E2 -27582.007} C_VEL
LIN {X 0,Y 117.39,Z 285.802,A -85,B 0,C 180,E1 -27586.939,E2 -27586.939} C_VEL
LIN {X 0,Y 116.574,Z 292.941,A -85,B 0,C 180,E1 -27592.924,E2 -27592.924} C_VEL
LIN {X 0,Y 116.798,Z 297.428,A -85,B 0,C 180,E1 -27597.392,E2 -27597.392} C_VEL
LIN {X 0,Y 118.244,Z 302.133,A -85,B 0,C 180,E1 -27603.063,E2 -27603.063} C_VEL
LIN {X 0,Y 121.023,Z 305.753,A -85,B 0,C 180,E1 -27608.369,E2 -27608.369} C_VEL
LIN {X 0,Y 122.251,Z 307.344,A -85,B 0,C 180,E1 -27611.004,E2 -27611.004} C_VEL
LIN {X 0,Y 123.246,Z 309.813,A -85,B 0,C 180,E1 -27615.472,E2 -27615.472} C_VEL
LIN {X 0,Y 124.58,Z 311.364,A -85,B 0,C 180,E1 -27618.995,E2 -27618.995} C_VEL
LIN {X 0,Y 126.692,Z 312.144,A -85,B 0,C 180,E1 -27621.465,E2 -27621.465} C_VEL
LIN {X 0,Y 127.695,Z 312.317,A -85,B 0,C 180,E1 -27622.217,E2 -27622.217} C_VEL
LIN {X 0,Y 135.954,Z 313.041,A -85,B 0,C 180,E1 -27627.037,E2 -27627.037} C_VEL
LIN {X 0,Y 142.234,Z 313.001,A -85,B 0,C 180,E1 -27630,E2 -27630} C_VEL
LIN {X 0,Y 133.865,Z 312.904,A -85,B 0,C 180,E1 -27634.067,E2 -27634.067} C_VEL
LIN {X 0,Y 124.938,Z 311.785,A -85,B 0,C 180,E1 -27639.715,E2 -27639.715} C_VEL
LIN {X 0,Y 120.446,Z 310.589,A -85,B 0,C 180,E1 -27643.497,E2 -27643.497} C_VEL
LIN {X 0,Y 115.068,Z 307.924,A -85,B 0,C 180,E1 -27649.628,E2 -27649.628} C_VEL
LIN {X 0,Y 112.543,Z 305.651,A -85,B 0,C 180,E1 -27653.946,E2 -27653.946} C_VEL
LIN {X 0,Y 110.347,Z 301.171,A -85,B 0,C 180,E1 -27660.631,E2 -27660.631} C_VEL
LIN {X 0,Y 109.915,Z 295.41,A -85,B 0,C 180,E1 -27667.404,E2 -27667.404} C_VEL
LIN {X 0,Y 110.847,Z 289.53,A -85,B 0,C 180,E1 -27672.965,E2 -27672.965} C_VEL
LIN {X 0,Y 111.43,Z 284.746,A -85,B 0,C 180,E1 -27677.217,E2 -27677.217} C_VEL
LIN {X 0,Y 111.589,Z 279.154,A -85,B 0,C 180,E1 -27682.12,E2 -27682.12} C_VEL
LIN {X 0,Y 111.263,Z 274.733,A -85,B 0,C 180,E1 -27686.181,E2 -27686.181} C_VEL
LIN {X 0,Y 110.624,Z 269.476,A -85,B 0,C 180,E1 -27691.549,E2 -27691.549} C_VEL
LIN {X 0,Y 109.971,Z 266.114,A -85,B 0,C 180,E1 -27695.458,E2 -27695.458} C_VEL
LIN {X 0,Y 108.989,Z 262.163,A -85,B 0,C 180,E1 -27701.193,E2 -27701.193} C_VEL
LIN {X 0,Y 108.072,Z 259.049,A -85,B 0,C 180,E1 -27707.278,E2 -27707.278} C_VEL
LIN {X 0,Y 107.587,Z 257.425,A -85,B 0,C 180,E1 -27712.495,E2 -27712.495} C_VEL
LIN {X 0,Y 107.979,Z 255.774,A -85,B 0,C 180,E1 -27720.002,E2 -27720.002} C_VEL
LIN {X 0,Y 107.91,Z 257.763,A -85,B 0,C 180,E1 -27727.486,E2 -27727.486} C_VEL
LIN {X 0,Y 108.357,Z 259.053,A -85,B 0,C 180,E1 -27731.222,E2 -27731.222} C_VEL
LIN {X 0,Y 108.918,Z 262.53,A -85,B 0,C 180,E1 -27736.882,E2 -27736.882} C_VEL
LIN {X 0,Y 109.384,Z 265.628,A -85,B 0,C 180,E1 -27740.696,E2 -27740.696} C_VEL
LIN {X 0,Y 109.711,Z 271.482,A -85,B 0,C 180,E1 -27746.644,E2 -27746.644} C_VEL
LIN {X 0,Y 109.68,Z 275.191,A -85,B 0,C 180,E1 -27749.777,E2 -27749.777} C_VEL
LIN {X 0,Y 109.067,Z 278.373,A -85,B 0,C 180,E1 -27752.121,E2 -27752.121} C_VEL
LIN {X 0,Y 107.562,Z 283.066,A -85,B 0,C 180,E1 -27755.063,E2 -27755.063} C_VEL
LIN {X 0,Y 104.741,Z 289.808,A -85,B 0,C 180,E1 -27759.5,E2 -27759.5} C_VEL
LIN {X 0,Y 103.273,Z 292.61,A -85,B 0,C 180,E1 -27761.533,E2 -27761.533} C_VEL
LIN {X 0,Y 98.867,Z 297.779,A -85,B 0,C 180,E1 -27764.696,E2 -27764.696} C_VEL
LIN {X 0,Y 94.686,Z 302.285,A -85,B 0,C 180,E1 -27768.087,E2 -27768.087} C_VEL
LIN {X 0,Y 89.001,Z 307.781,A -85,B 0,C 180,E1 -27773.684,E2 -27773.684} C_VEL
LIN {X 0,Y 84.23,Z 312.112,A -85,B 0,C 180,E1 -27779.959,E2 -27779.959} C_VEL
LIN {X 0,Y 81.589,Z 314.483,A -85,B 0,C 180,E1 -27784.489,E2 -27784.489} C_VEL
LIN {X 0,Y 79.592,Z 316.291,A -85,B 0,C 180,E1 -27789.317,E2 -27789.317} C_VEL
LIN {X 0,Y 77.183,Z 318.758,A -85,B 0,C 180,E1 -27799.507,E2 -27799.507} C_VEL
LIN {X 0,Y 76.739,Z 319.357,A -85,B 0,C 180,E1 -27804.745,E2 -27804.745} C_VEL
LIN {X 0,Y 76.782,Z 319.52,A -85,B 0,C 180,E1 -27810,E2 -27810} C_VEL
LIN {X 0,Y 76.739,Z 319.357,A -85,B 0,C 180,E1 -27815.255,E2 -27815.255} C_VEL
LIN {X 0,Y 77.183,Z 318.758,A -85,B 0,C 180,E1 -27820.493,E2 -27820.493} C_VEL
LIN {X 0,Y 79.592,Z 316.291,A -85,B 0,C 180,E1 -27830.683,E2 -27830.683} C_VEL
LIN {X 0,Y 82.849,Z 313.331,A -85,B 0,C 180,E1 -27837.811,E2 -27837.811} C_VEL
LIN {X 0,Y 87.294,Z 309.336,A -85,B 0,C 180,E1 -27844.302,E2 -27844.302} C_VEL
LIN {X 0,Y 92.754,Z 304.204,A -85,B 0,C 180,E1 -27850.093,E2 -27850.093} C_VEL
LIN {X 0,Y 97.683,Z 299.051,A -85,B 0,C 180,E1 -27854.401,E2 -27854.401} C_VEL
LIN {X 0,Y 102.224,Z 293.992,A -85,B 0,C 180,E1 -27857.652,E2 -27857.652} C_VEL
LIN {X 0,Y 104,Z 291.213,A -85,B 0,C 180,E1 -27859.484,E2 -27859.484} C_VEL
LIN {X 0,Y 106.846,Z 284.892,A -85,B 0,C 180,E1 -27863.699,E2 -27863.699} C_VEL
LIN {X 0,Y 108.722,Z 279.5,A -85,B 0,C 180,E1 -27867.175,E2 -27867.175} C_VEL
LIN {X 0,Y 109.481,Z 276.614,A -85,B 0,C 180,E1 -27869.097,E2 -27869.097} C_VEL
LIN {X 0,Y 109.751,Z 272.637,A -85,B 0,C 180,E1 -27872.335,E2 -27872.335} C_VEL
LIN {X 0,Y 109.451,Z 267.486,A -85,B 0,C 180,E1 -27877.338,E2 -27877.338} C_VEL
LIN {X 0,Y 109.382,Z 265.631,A -85,B 0,C 180,E1 -27879.303,E2 -27879.303} C_VEL
LIN {X 0,Y 108.952,Z 262.476,A -85,B 0,C 180,E1 -27883.124,E2 -27883.124} C_VEL
LIN {X 0,Y 108.37,Z 259.033,A -85,B 0,C 180,E1 -27888.779,E2 -27888.779} C_VEL
LIN {X 0,Y 107.737,Z 256.756,A -85,B 0,C 180,E1 -27896.258,E2 -27896.258} C_VEL
LIN {X 0,Y 107.981,Z 255.77,A -85,B 0,C 180,E1 -27899.998,E2 -27899.998} C_VEL
LIN {X 0,Y 107.595,Z 257.442,A -85,B 0,C 180,E1 -27907.595,E2 -27907.595} C_VEL
LIN {X 0,Y 108.05,Z 259.051,A -85,B 0,C 180,E1 -27912.672,E2 -27912.672} C_VEL
LIN {X 0,Y 108.989,Z 262.162,A -85,B 0,C 180,E1 -27918.807,E2 -27918.807} C_VEL
LIN {X 0,Y 109.698,Z 264.627,A -85,B 0,C 180,E1 -27922.604,E2 -27922.604} C_VEL
LIN {X 0,Y 110.394,Z 268.103,A -85,B 0,C 180,E1 -27926.968,E2 -27926.968} C_VEL
LIN {X 0,Y 110.934,Z 271.41,A -85,B 0,C 180,E1 -27930.45,E2 -27930.45} C_VEL
LIN {X 0,Y 111.452,Z 276.714,A -85,B 0,C 180,E1 -27935.677,E2 -27935.677} C_VEL
LIN {X 0,Y 111.576,Z 281.392,A -85,B 0,C 180,E1 -27939.937,E2 -27939.937} C_VEL
LIN {X 0,Y 111.157,Z 287.298,A -85,B 0,C 180,E1 -27945.07,E2 -27945.07} C_VEL
LIN {X 0,Y 110.202,Z 293.183,A -85,B 0,C 180,E1 -27950.377,E2 -27950.377} C_VEL
LIN {X 0,Y 109.929,Z 298.615,A -85,B 0,C 180,E1 -27956.21,E2 -27956.21} C_VEL
LIN {X 0,Y 111.069,Z 303.233,A -85,B 0,C 180,E1 -27962.353,E2 -27962.353} C_VEL
LIN {X 0,Y 113.715,Z 306.799,A -85,B 0,C 180,E1 -27968.234,E2 -27968.234} C_VEL
LIN {X 0,Y 117.395,Z 309.303,A -85,B 0,C 180,E1 -27973.301,E2 -27973.301} C_VEL
LIN {X 0,Y 122.131,Z 311.175,A -85,B 0,C 180,E1 -27978.021,E2 -27978.021} C_VEL
LIN {X 0,Y 127.695,Z 312.317,A -85,B 0,C 180,E1 -27982.217,E2 -27982.217} C_VEL
LIN {X 0,Y 128.441,Z 312.649,A -85,B 0,C 180,E1 -27983.436,E2 -27983.436} C_VEL
LIN {X 0,Y 127.741,Z 313.325,A -85,B 0,C 180,E1 -27987.035,E2 -27987.035} C_VEL
LIN {X 0,Y 128.67,Z 313.324,A -85,B 0,C 180,E1 -27988.036,E2 -27988.036} C_VEL
LIN {X 0,Y 132.587,Z 313.288,A -85,B 0,C 180,E1 -27990,E2 -27990} C_VEL
LIN {X 0,Y 126.421,Z 313.326,A -85,B 0,C 180,E1 -27993.187,E2 -27993.187} C_VEL
LIN {X 0,Y 120.362,Z 312.897,A -85,B 0,C 180,E1 -27996.972,E2 -27996.972} C_VEL
LIN {X 0,Y 111.651,Z 310.859,A -85,B 0,C 180,E1 -28004.583,E2 -28004.583} C_VEL
LIN {X 0,Y 108.186,Z 309.246,A -85,B 0,C 180,E1 -28008.954,E2 -28008.954} C_VEL
LIN {X 0,Y 104.753,Z 305.905,A -85,B 0,C 180,E1 -28015.855,E2 -28015.855} C_VEL
LIN {X 0,Y 103.187,Z 301.422,A -85,B 0,C 180,E1 -28023.016,E2 -28023.016} C_VEL
LIN {X 0,Y 103.525,Z 295.907,A -85,B 0,C 180,E1 -28029.869,E2 -28029.869} C_VEL
LIN {X 0,Y 104.656,Z 291.103,A -85,B 0,C 180,E1 -28034.838,E2 -28034.838} C_VEL
LIN {X 0,Y 105.552,Z 285.033,A -85,B 0,C 180,E1 -28040.768,E2 -28040.768} C_VEL
LIN {X 0,Y 105.731,Z 281.025,A -85,B 0,C 180,E1 -28044.698,E2 -28044.698} C_VEL
LIN {X 0,Y 105.566,Z 276.172,A -85,B 0,C 180,E1 -28049.935,E2 -28049.935} C_VEL
LIN {X 0,Y 105.344,Z 272.508,A -85,B 0,C 180,E1 -28054.303,E2 -28054.303} C_VEL
LIN {X 0,Y 104.611,Z 268.362,A -85,B 0,C 180,E1 -28060.374,E2 -28060.374} C_VEL
LIN {X 0,Y 104.228,Z 266.211,A -85,B 0,C 180,E1 -28064.355,E2 -28064.355} C_VEL
LIN {X 0,Y 103.952,Z 264.581,A -85,B 0,C 180,E1 -28068.3,E2 -28068.3} C_VEL
LIN {X 0,Y 103.676,Z 262.588,A -85,B 0,C 180,E1 -28076.115,E2 -28076.115} C_VEL
LIN {X 0,Y 104.089,Z 261.797,A -85,B 0,C 180,E1 -28080.002,E2 -28080.002} C_VEL
LIN {X 0,Y 103.989,Z 263.835,A -85,B 0,C 180,E1 -28087.77,E2 -28087.77} C_VEL
LIN {X 0,Y 104.321,Z 265.327,A -85,B 0,C 180,E1 -28091.662,E2 -28091.662} C_VEL
LIN {X 0,Y 104.458,Z 267.58,A -85,B 0,C 180,E1 -28095.614,E2 -28095.614} C_VEL
LIN {X 0,Y 104.585,Z 270.648,A -85,B 0,C 180,E1 -28099.819,E2 -28099.819} C_VEL
LIN {X 0,Y 104.539,Z 275.386,A -85,B 0,C 180,E1 -28105.008,E2 -28105.008} C_VEL
LIN {X 0,Y 104.144,Z 279.234,A -85,B 0,C 180,E1 -28108.685,E2 -28108.685} C_VEL
LIN {X 0,Y 103.665,Z 281.215,A -85,B 0,C 180,E1 -28110.192,E2 -28110.192} C_VEL
LIN {X 0,Y 100.486,Z 288.493,A -85,B 0,C 180,E1 -28115.274,E2 -28115.274} C_VEL
LIN {X 0,Y 97.512,Z 293.777,A -85,B 0,C 180,E1 -28119.216,E2 -28119.216} C_VEL
LIN {X 0,Y 91.485,Z 300.111,A -85,B 0,C 180,E1 -28123.452,E2 -28123.452} C_VEL
LIN {X 0,Y 85.374,Z 305.909,A -85,B 0,C 180,E1 -28128.81,E2 -28128.81} C_VEL
LIN {X 0,Y 79.775,Z 310.657,A -85,B 0,C 180,E1 -28135.066,E2 -28135.066} C_VEL
LIN {X 0,Y 75.213,Z 314.27,A -85,B 0,C 180,E1 -28142.147,E2 -28142.147} C_VEL
LIN {X 0,Y 72.959,Z 316.079,A -85,B 0,C 180,E1 -28147.337,E2 -28147.337} C_VEL
LIN {X 0,Y 70.193,Z 318.546,A -85,B 0,C 180,E1 -28158.449,E2 -28158.449} C_VEL
LIN {X 0,Y 69.655,Z 319.145,A -85,B 0,C 180,E1 -28164.209,E2 -28164.209} C_VEL
LIN {X 0,Y 69.703,Z 319.309,A -85,B 0,C 180,E1 -28170,E2 -28170} C_VEL
LIN {X 0,Y 69.655,Z 319.145,A -85,B 0,C 180,E1 -28175.791,E2 -28175.791} C_VEL
LIN {X 0,Y 70.193,Z 318.546,A -85,B 0,C 180,E1 -28181.551,E2 -28181.551} C_VEL
LIN {X 0,Y 72.959,Z 316.079,A -85,B 0,C 180,E1 -28192.663,E2 -28192.663} C_VEL
LIN {X 0,Y 76.618,Z 313.119,A -85,B 0,C 180,E1 -28200.298,E2 -28200.298} C_VEL
LIN {X 0,Y 81.493,Z 309.124,A -85,B 0,C 180,E1 -28207.134,E2 -28207.134} C_VEL
LIN {X 0,Y 87.409,Z 303.991,A -85,B 0,C 180,E1 -28213.111,E2 -28213.111} C_VEL
LIN {X 0,Y 92.707,Z 298.838,A -85,B 0,C 180,E1 -28217.496,E2 -28217.496} C_VEL
LIN {X 0,Y 97.476,Z 293.775,A -85,B 0,C 180,E1 -28220.81,E2 -28220.81} C_VEL
LIN {X 0,Y 100.494,Z 288.469,A -85,B 0,C 180,E1 -28224.744,E2 -28224.744} C_VEL
LIN {X 0,Y 103.666,Z 281.189,A -85,B 0,C 180,E1 -28229.831,E2 -28229.831} C_VEL
LIN {X 0,Y 104.372,Z 277.572,A -85,B 0,C 180,E1 -28232.796,E2 -28232.796} C_VEL
LIN {X 0,Y 104.61,Z 274.222,A -85,B 0,C 180,E1 -28236.226,E2 -28236.226} C_VEL
LIN {X 0,Y 104.587,Z 270.49,A -85,B 0,C 180,E1 -28240.365,E2 -28240.365} C_VEL
LIN {X 0,Y 104.5,Z 267.523,A -85,B 0,C 180,E1 -28244.392,E2 -28244.392} C_VEL
LIN {X 0,Y 104.334,Z 265.308,A -85,B 0,C 180,E1 -28248.339,E2 -28248.339} C_VEL
LIN {X 0,Y 104.006,Z 263.808,A -85,B 0,C 180,E1 -28252.231,E2 -28252.231} C_VEL
LIN {X 0,Y 104.086,Z 261.802,A -85,B 0,C 180,E1 -28259.998,E2 -28259.998} C_VEL
LIN {X 0,Y 103.685,Z 263.466,A -85,B 0,C 180,E1 -28267.789,E2 -28267.789} C_VEL
LIN {X 0,Y 103.942,Z 264.595,A -85,B 0,C 180,E1 -28271.701,E2 -28271.701} C_VEL
LIN {X 0,Y 104.405,Z 267.221,A -85,B 0,C 180,E1 -28277.631,E2 -28277.631} C_VEL
LIN {X 0,Y 105.161,Z 270.979,A -85,B 0,C 180,E1 -28283.637,E2 -28283.637} C_VEL
LIN {X 0,Y 105.445,Z 274.209,A -85,B 0,C 180,E1 -28287.809,E2 -28287.809} C_VEL
LIN {X 0,Y 105.759,Z 279.518,A -85,B 0,C 180,E1 -28293.686,E2 -28293.686} C_VEL
LIN {X 0,Y 105.667,Z 283.658,A -85,B 0,C 180,E1 -28297.963,E2 -28297.963} C_VEL
LIN {X 0,Y 105.07,Z 288.455,A -85,B 0,C 180,E1 -28302.628,E2 -28302.628} C_VEL
LIN {X 0,Y 104.389,Z 292.311,A -85,B 0,C 180,E1 -28306.364,E2 -28306.364} C_VEL
LIN {X 0,Y 103.146,Z 299.028,A -85,B 0,C 180,E1 -28313.87,E2 -28313.87} C_VEL
LIN {X 0,Y 103.479,Z 302.998,A -85,B 0,C 180,E1 -28319.38,E2 -28319.38} C_VEL
LIN {X 0,Y 105.618,Z 307.06,A -85,B 0,C 180,E1 -28326.469,E2 -28326.469} C_VEL
LIN {X 0,Y 109.976,Z 310.119,A -85,B 0,C 180,E1 -28333.443,E2 -28333.443} C_VEL
LIN {X 0,Y 115.797,Z 312.061,A -85,B 0,C 180,E1 -28339.509,E2 -28339.509} C_VEL
LIN {X 0,Y 121.896,Z 313.008,A -85,B 0,C 180,E1 -28344.047,E2 -28344.047} C_VEL
LIN {X 0,Y 128.67,Z 313.324,A -85,B 0,C 180,E1 -28348.036,E2 -28348.036} C_VEL
LIN {X 0,Y 129.071,Z 313.394,A -85,B 0,C 180,E1 -28348.788,E2 -28348.788} C_VEL
LIN {X 0,Y 128.212,Z 313.419,A -85,B 0,C 180,E1 -28349.802,E2 -28349.802} C_VEL
LIN {X 0,Y 125.67,Z 313.506,A -85,B 0,C 180,E1 -28351.077,E2 -28351.077} C_VEL
LIN {X 0,Y 115.703,Z 313.497,A -85,B 0,C 180,E1 -28354.43,E2 -28354.43} C_VEL
LIN {X 0,Y 114.059,Z 313.4,A -85,B 0,C 180,E1 -28355.37,E2 -28355.37} C_VEL
LIN {X 0,Y 106.837,Z 312.333,A -85,B 0,C 180,E1 -28361.382,E2 -28361.382} C_VEL
LIN {X 0,Y 102.542,Z 310.949,A -85,B 0,C 180,E1 -28366.365,E2 -28366.365} C_VEL
LIN {X 0,Y 98.921,Z 308.679,A -85,B 0,C 180,E1 -28372.547,E2 -28372.547} C_VEL
LIN {X 0,Y 96.611,Z 304.715,A -85,B 0,C 180,E1 -28380.611,E2 -28380.611} C_VEL
LIN {X 0,Y 96.306,Z 301.038,A -85,B 0,C 180,E1 -28386.612,E2 -28386.612} C_VEL
LIN {X 0,Y 97.734,Z 295.161,A -85,B 0,C 180,E1 -28394.024,E2 -28394.024} C_VEL
LIN {X 0,Y 98.998,Z 290.441,A -85,B 0,C 180,E1 -28399.261,E2 -28399.261} C_VEL
LIN {X 0,Y 99.768,Z 286.054,A -85,B 0,C 180,E1 -28404.142,E2 -28404.142} C_VEL
LIN {X 0,Y 100.031,Z 281.261,A -85,B 0,C 180,E1 -28409.712,E2 -28409.712} C_VEL
LIN {X 0,Y 100.109,Z 277.108,A -85,B 0,C 180,E1 -28415.091,E2 -28415.091} C_VEL
LIN {X 0,Y 99.918,Z 274.334,A -85,B 0,C 180,E1 -28419.412,E2 -28419.412} C_VEL
LIN {X 0,Y 99.735,Z 272.178,A -85,B 0,C 180,E1 -28423.631,E2 -28423.631} C_VEL
LIN {X 0,Y 99.505,Z 270.438,A -85,B 0,C 180,E1 -28427.769,E2 -28427.769} C_VEL
LIN {X 0,Y 99.35,Z 269.183,A -85,B 0,C 180,E1 -28432.029,E2 -28432.029} C_VEL
LIN {X 0,Y 99.923,Z 267.619,A -85,B 0,C 180,E1 -28440.002,E2 -28440.002} C_VEL
LIN {X 0,Y 99.678,Z 270.068,A -85,B 0,C 180,E1 -28449.22,E2 -28449.22} C_VEL
LIN {X 0,Y 99.816,Z 271.286,A -85,B 0,C 180,E1 -28452.197,E2 -28452.197} C_VEL
LIN {X 0,Y 99.702,Z 274.862,A -85,B 0,C 180,E1 -28457.945,E2 -28457.945} C_VEL
LIN {X 0,Y 99.291,Z 278.903,A -85,B 0,C 180,E1 -28463.052,E2 -28463.052} C_VEL
LIN {X 0,Y 98.89,Z 281.883,A -85,B 0,C 180,E1 -28466.216,E2 -28466.216} C_VEL
LIN {X 0,Y 97.801,Z 284.739,A -85,B 0,C 180,E1 -28468.742,E2 -28468.742} C_VEL
LIN {X 0,Y 94.471,Z 290.964,A -85,B 0,C 180,E1 -28473.483,E2 -28473.483} C_VEL
LIN {X 0,Y 91.92,Z 294.943,A -85,B 0,C 180,E1 -28476.602,E2 -28476.602} C_VEL
LIN {X 0,Y 84.43,Z 302.007,A -85,B 0,C 180,E1 -28481.757,E2 -28481.757} C_VEL
LIN {X 0,Y 77.986,Z 307.357,A -85,B 0,C 180,E1 -28487.478,E2 -28487.478} C_VEL
LIN {X 0,Y 72.239,Z 311.687,A -85,B 0,C 180,E1 -28494.287,E2 -28494.287} C_VEL
LIN {X 0,Y 68.989,Z 314.058,A -85,B 0,C 180,E1 -28499.38,E2 -28499.38} C_VEL
LIN {X 0,Y 66.438,Z 315.867,A -85,B 0,C 180,E1 -28504.968,E2 -28504.968} C_VEL
LIN {X 0,Y 63.221,Z 318.334,A -85,B 0,C 180,E1 -28517.154,E2 -28517.154} C_VEL
LIN {X 0,Y 62.585,Z 318.933,A -85,B 0,C 180,E1 -28523.552,E2 -28523.552} C_VEL
LIN {X 0,Y 62.613,Z 319.098,A -85,B 0,C 180,E1 -28530,E2 -28530} C_VEL
LIN {X 0,Y 62.585,Z 318.933,A -85,B 0,C 180,E1 -28536.448,E2 -28536.448} C_VEL
LIN {X 0,Y 63.221,Z 318.334,A -85,B 0,C 180,E1 -28542.846,E2 -28542.846} C_VEL
LIN {X 0,Y 66.438,Z 315.867,A -85,B 0,C 180,E1 -28555.032,E2 -28555.032} C_VEL
LIN {X 0,Y 70.56,Z 312.907,A -85,B 0,C 180,E1 -28563.217,E2 -28563.217} C_VEL
LIN {X 0,Y 75.926,Z 308.911,A -85,B 0,C 180,E1 -28570.386,E2 -28570.386} C_VEL
LIN {X 0,Y 81.694,Z 304.34,A -85,B 0,C 180,E1 -28575.943,E2 -28575.943} C_VEL
LIN {X 0,Y 88.165,Z 298.51,A -85,B 0,C 180,E1 -28581.005,E2 -28581.005} C_VEL
LIN {X 0,Y 91.878,Z 294.941,A -85,B 0,C 180,E1 -28583.433,E2 -28583.433} C_VEL
LIN {X 0,Y 95.224,Z 289.758,A -85,B 0,C 180,E1 -28587.493,E2 -28587.493} C_VEL
LIN {X 0,Y 97.811,Z 284.714,A -85,B 0,C 180,E1 -28591.279,E2 -28591.279} C_VEL
LIN {X 0,Y 98.907,Z 281.863,A -85,B 0,C 180,E1 -28593.789,E2 -28593.789} C_VEL
LIN {X 0,Y 99.307,Z 278.905,A -85,B 0,C 180,E1 -28596.927,E2 -28596.927} C_VEL
LIN {X 0,Y 99.699,Z 274.867,A -85,B 0,C 180,E1 -28602.051,E2 -28602.051} C_VEL
LIN {X 0,Y 99.862,Z 272.393,A -85,B 0,C 180,E1 -28605.738,E2 -28605.738} C_VEL
LIN {X 0,Y 99.71,Z 270.074,A -85,B 0,C 180,E1 -28610.668,E2 -28610.668} C_VEL
LIN {X 0,Y 99.914,Z 267.631,A -85,B 0,C 180,E1 -28619.998,E2 -28619.998} C_VEL
LIN {X 0,Y 99.342,Z 269.235,A -85,B 0,C 180,E1 -28628.132,E2 -28628.132} C_VEL
LIN {X 0,Y 99.489,Z 270.46,A -85,B 0,C 180,E1 -28632.233,E2 -28632.233} C_VEL
LIN {X 0,Y 99.811,Z 273.205,A -85,B 0,C 180,E1 -28638.471,E2 -28638.471} C_VEL
LIN {X 0,Y 100.032,Z 275.616,A -85,B 0,C 180,E1 -28642.731,E2 -28642.731} C_VEL
LIN {X 0,Y 100.145,Z 278.816,A -85,B 0,C 180,E1 -28647.137,E2 -28647.137} C_VEL
LIN {X 0,Y 99.914,Z 284.577,A -85,B 0,C 180,E1 -28654.242,E2 -28654.242} C_VEL
LIN {X 0,Y 99.311,Z 288.717,A -85,B 0,C 180,E1 -28658.883,E2 -28658.883} C_VEL
LIN {X 0,Y 98.189,Z 293.668,A -85,B 0,C 180,E1 -28664.295,E2 -28664.295} C_VEL
LIN {X 0,Y 96.522,Z 299.734,A -85,B 0,C 180,E1 -28671.616,E2 -28671.616} C_VEL
LIN {X 0,Y 96.611,Z 304.715,A -85,B 0,C 180,E1 -28679.389,E2 -28679.389} C_VEL
LIN {X 0,Y 98.922,Z 308.679,A -85,B 0,C 180,E1 -28687.452,E2 -28687.452} C_VEL
LIN {X 0,Y 102.962,Z 311.127,A -85,B 0,C 180,E1 -28694.155,E2 -28694.155} C_VEL
LIN {X 0,Y 111.512,Z 313.207,A -85,B 0,C 180,E1 -28702.759,E2 -28702.759} C_VEL
LIN {X 0,Y 119.538,Z 313.679,A -85,B 0,C 180,E1 -28708.09,E2 -28708.09} C_VEL
LIN {X 0,Y 123.017,Z 313.573,A -85,B 0,C 180,E1 -28710,E2 -28710} C_VEL
LIN {X 0,Y 114.059,Z 313.4,A -85,B 0,C 180,E1 -28715.37,E2 -28715.37} C_VEL
LIN {X 0,Y 110.199,Z 313.196,A -85,B 0,C 180,E1 -28717.66,E2 -28717.66} C_VEL
LIN {X 0,Y 97.513,Z 312.098,A -85,B 0,C 180,E1 -28724.558,E2 -28724.558} C_VEL
LIN {X 0,Y 94.426,Z 311.326,A -85,B 0,C 180,E1 -28727.504,E2 -28727.504} C_VEL
LIN {X 0,Y 93.711,Z 310.982,A -85,B 0,C 180,E1 -28728.595,E2 -28728.595} C_VEL
LIN {X 0,Y 90.91,Z 308.702,A -85,B 0,C 180,E1 -28735.16,E2 -28735.16} C_VEL
LIN {X 0,Y 89.738,Z 306.452,A -85,B 0,C 180,E1 -28740.521,E2 -28740.521} C_VEL
LIN {X 0,Y 89.74,Z 301.915,A -85,B 0,C 180,E1 -28748.793,E2 -28748.793} C_VEL
LIN {X 0,Y 91.614,Z 296.445,A -85,B 0,C 180,E1 -28756.34,E2 -28756.34} C_VEL
LIN {X 0,Y 93.045,Z 292.18,A -85,B 0,C 180,E1 -28761.69,E2 -28761.69} C_VEL
LIN {X 0,Y 94.011,Z 287.747,A -85,B 0,C 180,E1 -28767.157,E2 -28767.157} C_VEL
LIN {X 0,Y 94.515,Z 283.157,A -85,B 0,C 180,E1 -28773.506,E2 -28773.506} C_VEL
LIN {X 0,Y 94.801,Z 280.173,A -85,B 0,C 180,E1 -28778.246,E2 -28778.246} C_VEL
LIN {X 0,Y 94.779,Z 277.833,A -85,B 0,C 180,E1 -28782.749,E2 -28782.749} C_VEL
LIN {X 0,Y 94.718,Z 276.053,A -85,B 0,C 180,E1 -28787.141,E2 -28787.141} C_VEL
LIN {X 0,Y 94.725,Z 274.808,A -85,B 0,C 180,E1 -28791.469,E2 -28791.469} C_VEL
LIN {X 0,Y 95.478,Z 273.259,A -85,B 0,C 180,E1 -28800.002,E2 -28800.002} C_VEL
LIN {X 0,Y 95.038,Z 275.302,A -85,B 0,C 180,E1 -28808.508,E2 -28808.508} C_VEL
LIN {X 0,Y 94.943,Z 277.057,A -85,B 0,C 180,E1 -28812.833,E2 -28812.833} C_VEL
LIN {X 0,Y 94.543,Z 279.777,A -85,B 0,C 180,E1 -28817.301,E2 -28817.301} C_VEL
LIN {X 0,Y 93.672,Z 283.951,A -85,B 0,C 180,E1 -28822.937,E2 -28822.937} C_VEL
LIN {X 0,Y 93.127,Z 285.822,A -85,B 0,C 180,E1 -28825.097,E2 -28825.097} C_VEL
LIN {X 0,Y 91.038,Z 289.64,A -85,B 0,C 180,E1 -28828.307,E2 -28828.307} C_VEL
LIN {X 0,Y 87.56,Z 294.715,A -85,B 0,C 180,E1 -28832.567,E2 -28832.567} C_VEL
LIN {X 0,Y 86.528,Z 295.986,A -85,B 0,C 180,E1 -28833.642,E2 -28833.642} C_VEL
LIN {X 0,Y 79.272,Z 302.245,A -85,B 0,C 180,E1 -28838.363,E2 -28838.363} C_VEL
LIN {X 0,Y 72.902,Z 307.145,A -85,B 0,C 180,E1 -28843.696,E2 -28843.696} C_VEL
LIN {X 0,Y 66.586,Z 311.475,A -85,B 0,C 180,E1 -28850.708,E2 -28850.708} C_VEL
LIN {X 0,Y 62.965,Z 313.846,A -85,B 0,C 180,E1 -28856.077,E2 -28856.077} C_VEL
LIN {X 0,Y 60.038,Z 315.654,A -85,B 0,C 180,E1 -28862.08,E2 -28862.08} C_VEL
LIN {X 0,Y 56.304,Z 318.122,A -85,B 0,C 180,E1 -28875.544,E2 -28875.544} C_VEL
LIN {X 0,Y 55.539,Z 318.722,A -85,B 0,C 180,E1 -28882.73,E2 -28882.73} C_VEL
LIN {X 0,Y 55.513,Z 318.887,A -85,B 0,C 180,E1 -28890,E2 -28890} C_VEL
LIN {X 0,Y 55.539,Z 318.722,A -85,B 0,C 180,E1 -28897.27,E2 -28897.27} C_VEL
LIN {X 0,Y 56.304,Z 318.122,A -85,B 0,C 180,E1 -28904.456,E2 -28904.456} C_VEL
LIN {X 0,Y 60.038,Z 315.654,A -85,B 0,C 180,E1 -28917.92,E2 -28917.92} C_VEL
LIN {X 0,Y 64.723,Z 312.695,A -85,B 0,C 180,E1 -28926.67,E2 -28926.67} C_VEL
LIN {X 0,Y 70.648,Z 308.699,A -85,B 0,C 180,E1 -28934.134,E2 -28934.134} C_VEL
LIN {X 0,Y 76.573,Z 304.392,A -85,B 0,C 180,E1 -28939.499,E2 -28939.499} C_VEL
LIN {X 0,Y 82.559,Z 299.454,A -85,B 0,C 180,E1 -28943.969,E2 -28943.969} C_VEL
LIN {X 0,Y 86.495,Z 295.984,A -85,B 0,C 180,E1 -28946.391,E2 -28946.391} C_VEL
LIN {X 0,Y 89.5,Z 291.915,A -85,B 0,C 180,E1 -28949.741,E2 -28949.741} C_VEL
LIN {X 0,Y 92.155,Z 287.817,A -85,B 0,C 180,E1 -28953.176,E2 -28953.176} C_VEL
LIN {X 0,Y 93.122,Z 285.822,A -85,B 0,C 180,E1 -28954.909,E2 -28954.909} C_VEL
LIN {X 0,Y 93.899,Z 283.165,A -85,B 0,C 180,E1 -28958.021,E2 -28958.021} C_VEL
LIN {X 0,Y 94.565,Z 279.752,A -85,B 0,C 180,E1 -28962.704,E2 -28962.704} C_VEL
LIN {X 0,Y 94.966,Z 277.032,A -85,B 0,C 180,E1 -28967.17,E2 -28967.17} C_VEL
LIN {X 0,Y 95.073,Z 275.263,A -85,B 0,C 180,E1 -28971.496,E2 -28971.496} C_VEL
LIN {X 0,Y 95.474,Z 273.264,A -85,B 0,C 180,E1 -28979.998,E2 -28979.998} C_VEL
LIN {X 0,Y 94.724,Z 274.81,A -85,B 0,C 180,E1 -28988.531,E2 -28988.531} C_VEL
LIN {X 0,Y 94.749,Z 276.999,A -85,B 0,C 180,E1 -28995.365,E2 -28995.365} C_VEL
LIN {X 0,Y 94.849,Z 278.916,A -85,B 0,C 180,E1 -28999.475,E2 -28999.475} C_VEL
LIN {X 0,Y 94.719,Z 281.521,A -85,B 0,C 180,E1 -29004.082,E2 -29004.082} C_VEL
LIN {X 0,Y 94.163,Z 286.781,A -85,B 0,C 180,E1 -29011.494,E2 -29011.494} C_VEL
LIN {X 0,Y 93.562,Z 290.022,A -85,B 0,C 180,E1 -29015.757,E2 -29015.757} C_VEL
LIN {X 0,Y 92.46,Z 293.921,A -85,B 0,C 180,E1 -29020.527,E2 -29020.527} C_VEL
LIN {X 0,Y 90.932,Z 298.243,A -85,B 0,C 180,E1 -29025.926,E2 -29025.926} C_VEL
LIN {X 0,Y 89.527,Z 303.58,A -85,B 0,C 180,E1 -29034.097,E2 -29034.097} C_VEL
LIN {X 0,Y 90.184,Z 307.569,A -85,B 0,C 180,E1 -29042.123,E2 -29042.123} C_VEL
LIN {X 0,Y 91.807,Z 309.767,A -85,B 0,C 180,E1 -29047.496,E2 -29047.496} C_VEL
LIN {X 0,Y 95.157,Z 311.735,A -85,B 0,C 180,E1 -29053.759,E2 -29053.759} C_VEL
LIN {X 0,Y 102.386,Z 313.481,A -85,B 0,C 180,E1 -29062.109,E2 -29062.109} C_VEL
LIN {X 0,Y 107.571,Z 313.888,A -85,B 0,C 180,E1 -29066.254,E2 -29066.254} C_VEL
LIN {X 0,Y 113.523,Z 313.856,A -85,B 0,C 180,E1 -29070,E2 -29070} C_VEL
LIN {X 0,Y 105.825,Z 313.757,A -85,B 0,C 180,E1 -29075.04,E2 -29075.04} C_VEL
LIN {X 0,Y 97.967,Z 312.603,A -85,B 0,C 180,E1 -29082.428,E2 -29082.428} C_VEL
LIN {X 0,Y 93.711,Z 310.982,A -85,B 0,C 180,E1 -29088.595,E2 -29088.595} C_VEL
LIN {X 0,Y 91.418,Z 310.039,A -85,B 0,C 180,E1 -29091.918,E2 -29091.918} C_VEL
LIN {X 0,Y 83.742,Z 306.959,A -85,B 0,C 180,E1 -29102.272,E2 -29102.272} C_VEL
LIN {X 0,Y 82.71,Z 305.408,A -85,B 0,C 180,E1 -29106.103,E2 -29106.103} C_VEL
LIN {X 0,Y 82.724,Z 304.779,A -85,B 0,C 180,E1 -29107.389,E2 -29107.389} C_VEL
LIN {X 0,Y 84.304,Z 300.322,A -85,B 0,C 180,E1 -29115.12,E2 -29115.12} C_VEL
LIN {X 0,Y 86.184,Z 296.329,A -85,B 0,C 180,E1 -29120.874,E2 -29120.874} C_VEL
LIN {X 0,Y 87.82,Z 291.81,A -85,B 0,C 180,E1 -29127.308,E2 -29127.308} C_VEL
LIN {X 0,Y 88.667,Z 288.011,A -85,B 0,C 180,E1 -29133.082,E2 -29133.082} C_VEL
LIN {X 0,Y 89.175,Z 285.79,A -85,B 0,C 180,E1 -29136.796,E2 -29136.796} C_VEL
LIN {X 0,Y 89.476,Z 283.245,A -85,B 0,C 180,E1 -29141.691,E2 -29141.691} C_VEL
LIN {X 0,Y 89.645,Z 281.439,A -85,B 0,C 180,E1 -29146.399,E2 -29146.399} C_VEL
LIN {X 0,Y 89.806,Z 280.182,A -85,B 0,C 180,E1 -29150.998,E2 -29150.998} C_VEL
LIN {X 0,Y 90.631,Z 278.543,A -85,B 0,C 180,E1 -29160.002,E2 -29160.002} C_VEL
LIN {X 0,Y 90.218,Z 279.501,A -85,B 0,C 180,E1 -29164.47,E2 -29164.47} C_VEL
LIN {X 0,Y 90.05,Z 280.773,A -85,B 0,C 180,E1 -29168.983,E2 -29168.983} C_VEL
LIN {X 0,Y 89.631,Z 282.709,A -85,B 0,C 180,E1 -29173.608,E2 -29173.608} C_VEL
LIN {X 0,Y 88.766,Z 285.611,A -85,B 0,C 180,E1 -29178.466,E2 -29178.466} C_VEL
LIN {X 0,Y 87.872,Z 288.432,A -85,B 0,C 180,E1 -29182.33,E2 -29182.33} C_VEL
LIN {X 0,Y 87.101,Z 289.755,A -85,B 0,C 180,E1 -29183.796,E2 -29183.796} C_VEL
LIN {X 0,Y 83.608,Z 294.482,A -85,B 0,C 180,E1 -29188.042,E2 -29188.042} C_VEL
LIN {X 0,Y 81.371,Z 296.93,A -85,B 0,C 180,E1 -29190.267,E2 -29190.267} C_VEL
LIN {X 0,Y 74.324,Z 302.554,A -85,B 0,C 180,E1 -29194.569,E2 -29194.569} C_VEL
LIN {X 0,Y 68.179,Z 306.934,A -85,B 0,C 180,E1 -29199.367,E2 -29199.367} C_VEL
LIN {X 0,Y 61.243,Z 311.264,A -85,B 0,C 180,E1 -29206.486,E2 -29206.486} C_VEL
LIN {X 0,Y 57.198,Z 313.634,A -85,B 0,C 180,E1 -29212.095,E2 -29212.095} C_VEL
LIN {X 0,Y 51.215,Z 316.839,A -85,B 0,C 180,E1 -29225.69,E2 -29225.69} C_VEL
LIN {X 0,Y 49.453,Z 317.91,A -85,B 0,C 180,E1 -29233.487,E2 -29233.487} C_VEL
LIN {X 0,Y 48.496,Z 318.51,A -85,B 0,C 180,E1 -29241.668,E2 -29241.668} C_VEL
LIN {X 0,Y 48.43,Z 318.676,A -85,B 0,C 180,E1 -29250,E2 -29250} C_VEL
LIN {X 0,Y 48.496,Z 318.51,A -85,B 0,C 180,E1 -29258.332,E2 -29258.332} C_VEL
LIN {X 0,Y 49.453,Z 317.91,A -85,B 0,C 180,E1 -29266.513,E2 -29266.513} C_VEL
LIN {X 0,Y 53.828,Z 315.441,A -85,B 0,C 180,E1 -29281.483,E2 -29281.483} C_VEL
LIN {X 0,Y 59.17,Z 312.483,A -85,B 0,C 180,E1 -29290.788,E2 -29290.788} C_VEL
LIN {X 0,Y 65.725,Z 308.487,A -85,B 0,C 180,E1 -29298.461,E2 -29298.461} C_VEL
LIN {X 0,Y 72.875,Z 303.609,A -85,B 0,C 180,E1 -29304.416,E2 -29304.416} C_VEL
LIN {X 0,Y 79.95,Z 298.085,A -85,B 0,C 180,E1 -29308.988,E2 -29308.988} C_VEL
LIN {X 0,Y 81.341,Z 296.928,A -85,B 0,C 180,E1 -29309.769,E2 -29309.769} C_VEL
LIN {X 0,Y 83.609,Z 294.482,A -85,B 0,C 180,E1 -29311.957,E2 -29311.957} C_VEL
LIN {X 0,Y 87.096,Z 289.76,A -85,B 0,C 180,E1 -29316.202,E2 -29316.202} C_VEL
LIN {X 0,Y 88.294,Z 287.341,A -85,B 0,C 180,E1 -29319.008,E2 -29319.008} C_VEL
LIN {X 0,Y 89.232,Z 284.154,A -85,B 0,C 180,E1 -29323.763,E2 -29323.763} C_VEL
LIN {X 0,Y 89.614,Z 282.725,A -85,B 0,C 180,E1 -29326.39,E2 -29326.39} C_VEL
LIN {X 0,Y 90.078,Z 280.744,A -85,B 0,C 180,E1 -29331.02,E2 -29331.02} C_VEL
LIN {X 0,Y 90.223,Z 279.495,A -85,B 0,C 180,E1 -29335.53,E2 -29335.53} C_VEL
LIN {X 0,Y 90.619,Z 278.556,A -85,B 0,C 180,E1 -29339.998,E2 -29339.998} C_VEL
LIN {X 0,Y 89.799,Z 280.19,A -85,B 0,C 180,E1 -29349.003,E2 -29349.003} C_VEL
LIN {X 0,Y 89.634,Z 281.449,A -85,B 0,C 180,E1 -29353.602,E2 -29353.602} C_VEL
LIN {X 0,Y 89.427,Z 283.761,A -85,B 0,C 180,E1 -29359.428,E2 -29359.428} C_VEL
LIN {X 0,Y 89.202,Z 285.762,A -85,B 0,C 180,E1 -29363.197,E2 -29363.197} C_VEL
LIN {X 0,Y 88.371,Z 289.298,A -85,B 0,C 180,E1 -29368.979,E2 -29368.979} C_VEL
LIN {X 0,Y 87.561,Z 292.831,A -85,B 0,C 180,E1 -29374.181,E2 -29374.181} C_VEL
LIN {X 0,Y 85.612,Z 297.761,A -85,B 0,C 180,E1 -29381.047,E2 -29381.047} C_VEL
LIN {X 0,Y 83.19,Z 303.18,A -85,B 0,C 180,E1 -29389.489,E2 -29389.489} C_VEL
LIN {X 0,Y 82.698,Z 307.361,A -85,B 0,C 180,E1 -29398.189,E2 -29398.189} C_VEL
LIN {X 0,Y 84.318,Z 310.365,A -85,B 0,C 180,E1 -29406.465,E2 -29406.465} C_VEL
LIN {X 0,Y 87.742,Z 312.416,A -85,B 0,C 180,E1 -29413.974,E2 -29413.974} C_VEL
LIN {X 0,Y 93.381,Z 313.752,A -85,B 0,C 180,E1 -29421.343,E2 -29421.343} C_VEL
LIN {X 0,Y 98.615,Z 314.182,A -85,B 0,C 180,E1 -29426.108,E2 -29426.108} C_VEL
LIN {X 0,Y 104.081,Z 314.137,A -85,B 0,C 180,E1 -29430,E2 -29430} C_VEL
LIN {X 0,Y 98.358,Z 314.162,A -85,B 0,C 180,E1 -29434.097,E2 -29434.097} C_VEL
LIN {X 0,Y 92.623,Z 313.671,A -85,B 0,C 180,E1 -29439.472,E2 -29439.472} C_VEL
LIN {X 0,Y 86.099,Z 311.653,A -85,B 0,C 180,E1 -29449.057,E2 -29449.057} C_VEL
LIN {X 0,Y 83.229,Z 308.956,A -85,B 0,C 180,E1 -29457.673,E2 -29457.673} C_VEL
LIN {X 0,Y 82.653,Z 305.213,A -85,B 0,C 180,E1 -29466.527,E2 -29466.527} C_VEL
LIN {X 0,Y 82.724,Z 304.779,A -85,B 0,C 180,E1 -29467.389,E2 -29467.389} C_VEL
LIN {X 0,Y 82.677,Z 302.985,A -85,B 0,C 180,E1 -29471.287,E2 -29471.287} C_VEL
LIN {X 0,Y 81.651,Z 300.062,A -85,B 0,C 180,E1 -29477.879,E2 -29477.879} C_VEL
LIN {X 0,Y 81.144,Z 296.376,A -85,B 0,C 180,E1 -29485.941,E2 -29485.941} C_VEL
LIN {X 0,Y 81.649,Z 294.856,A -85,B 0,C 180,E1 -29488.537,E2 -29488.537} C_VEL
LIN {X 0,Y 82.597,Z 292.392,A -85,B 0,C 180,E1 -29492.907,E2 -29492.907} C_VEL
LIN {X 0,Y 83.441,Z 289.638,A -85,B 0,C 180,E1 -29497.894,E2 -29497.894} C_VEL
LIN {X 0,Y 83.789,Z 288.467,A -85,B 0,C 180,E1 -29500.399,E2 -29500.399} C_VEL
LIN {X 0,Y 84.195,Z 286.611,A -85,B 0,C 180,E1 -29505.5,E2 -29505.5} C_VEL
LIN {X 0,Y 84.463,Z 285.195,A -85,B 0,C 180,E1 -29510.423,E2 -29510.423} C_VEL
LIN {X 0,Y 85.509,Z 283.563,A -85,B 0,C 180,E1 -29520.003,E2 -29520.003} C_VEL
LIN {X 0,Y 84.849,Z 284.924,A -85,B 0,C 180,E1 -29526.31,E2 -29526.31} C_VEL
LIN {X 0,Y 84.33,Z 286.882,A -85,B 0,C 180,E1 -29532.028,E2 -29532.028} C_VEL
LIN {X 0,Y 83.879,Z 288.149,A -85,B 0,C 180,E1 -29534.561,E2 -29534.561} C_VEL
LIN {X 0,Y 82.322,Z 291.414,A -85,B 0,C 180,E1 -29540.102,E2 -29540.102} C_VEL
LIN {X 0,Y 80.153,Z 294.243,A -85,B 0,C 180,E1 -29542.979,E2 -29542.979} C_VEL
LIN {X 0,Y 77.825,Z 296.704,A -85,B 0,C 180,E1 -29545.44,E2 -29545.44} C_VEL
LIN {X 0,Y 76.54,Z 297.874,A -85,B 0,C 180,E1 -29546.461,E2 -29546.461} C_VEL
LIN {X 0,Y 69.891,Z 302.772,A -85,B 0,C 180,E1 -29550.188,E2 -29550.188} C_VEL
LIN {X 0,Y 63.902,Z 306.722,A -85,B 0,C 180,E1 -29554.427,E2 -29554.427} C_VEL
LIN {X 0,Y 56.294,Z 311.052,A -85,B 0,C 180,E1 -29561.492,E2 -29561.492} C_VEL
LIN {X 0,Y 51.772,Z 313.423,A -85,B 0,C 180,E1 -29567.255,E2 -29567.255} C_VEL
LIN {X 0,Y 44.808,Z 316.627,A -85,B 0,C 180,E1 -29581.931,E2 -29581.931} C_VEL
LIN {X 0,Y 42.662,Z 317.698,A -85,B 0,C 180,E1 -29590.763,E2 -29590.763} C_VEL
LIN {X 0,Y 41.47,Z 318.299,A -85,B 0,C 180,E1 -29600.243,E2 -29600.243} C_VEL
LIN {X 0,Y 41.33,Z 318.465,A -85,B 0,C 180,E1 -29610,E2 -29610} C_VEL
LIN {X 0,Y 41.47,Z 318.299,A -85,B 0,C 180,E1 -29619.757,E2 -29619.757} C_VEL
LIN {X 0,Y 42.662,Z 317.698,A -85,B 0,C 180,E1 -29629.237,E2 -29629.237} C_VEL
LIN {X 0,Y 47.883,Z 315.229,A -85,B 0,C 180,E1 -29645.951,E2 -29645.951} C_VEL
LIN {X 0,Y 53.966,Z 312.271,A -85,B 0,C 180,E1 -29655.746,E2 -29655.746} C_VEL
LIN {X 0,Y 61.238,Z 308.275,A -85,B 0,C 180,E1 -29663.451,E2 -29663.451} C_VEL
LIN {X 0,Y 68.204,Z 303.918,A -85,B 0,C 180,E1 -29668.754,E2 -29668.754} C_VEL
LIN {X 0,Y 76.513,Z 297.872,A -85,B 0,C 180,E1 -29673.581,E2 -29673.581} C_VEL
LIN {X 0,Y 79,Z 295.525,A -85,B 0,C 180,E1 -29675.762,E2 -29675.762} C_VEL
LIN {X 0,Y 81.558,Z 292.491,A -85,B 0,C 180,E1 -29678.682,E2 -29678.682} C_VEL
LIN {X 0,Y 82.38,Z 291.31,A -85,B 0,C 180,E1 -29680.044,E2 -29680.044} C_VEL
LIN {X 0,Y 83.906,Z 288.126,A -85,B 0,C 180,E1 -29685.444,E2 -29685.444} C_VEL
LIN {X 0,Y 84.576,Z 285.928,A -85,B 0,C 180,E1 -29690.431,E2 -29690.431} C_VEL
LIN {X 0,Y 84.985,Z 284.524,A -85,B 0,C 180,E1 -29695.254,E2 -29695.254} C_VEL
LIN {X 0,Y 85.487,Z 283.583,A -85,B 0,C 180,E1 -29699.997,E2 -29699.997} C_VEL
LIN {X 0,Y 84.555,Z 284.777,A -85,B 0,C 180,E1 -29707.465,E2 -29707.465} C_VEL
LIN {X 0,Y 84.193,Z 286.613,A -85,B 0,C 180,E1 -29714.5,E2 -29714.5} C_VEL
LIN {X 0,Y 83.821,Z 288.441,A -85,B 0,C 180,E1 -29719.593,E2 -29719.593} C_VEL
LIN {X 0,Y 82.92,Z 291.241,A -85,B 0,C 180,E1 -29725.071,E2 -29725.071} C_VEL
LIN {X 0,Y 81.806,Z 294.57,A -85,B 0,C 180,E1 -29731.025,E2 -29731.025} C_VEL
LIN {X 0,Y 80.388,Z 297.75,A -85,B 0,C 180,E1 -29736.033,E2 -29736.033} C_VEL
LIN {X 0,Y 77.759,Z 302.398,A -85,B 0,C 180,E1 -29743.693,E2 -29743.693} C_VEL
LIN {X 0,Y 75.85,Z 306.909,A -85,B 0,C 180,E1 -29752.968,E2 -29752.968} C_VEL
LIN {X 0,Y 76.267,Z 310.277,A -85,B 0,C 180,E1 -29762.565,E2 -29762.565} C_VEL
LIN {X 0,Y 80.339,Z 313.017,A -85,B 0,C 180,E1 -29774.2,E2 -29774.2} C_VEL
LIN {X 0,Y 85.295,Z 314.095,A -85,B 0,C 180,E1 -29781.38,E2 -29781.38} C_VEL
LIN {X 0,Y 91.451,Z 314.515,A -85,B 0,C 180,E1 -29787.446,E2 -29787.446} C_VEL
LIN {X 0,Y 94.783,Z 314.414,A -85,B 0,C 180,E1 -29790,E2 -29790} C_VEL
LIN {X 0,Y 89.226,Z 314.435,A -85,B 0,C 180,E1 -29794.518,E2 -29794.518} C_VEL
LIN {X 0,Y 84.477,Z 314.02,A -85,B 0,C 180,E1 -29799.578,E2 -29799.578} C_VEL
LIN {X 0,Y 80.334,Z 313.021,A -85,B 0,C 180,E1 -29805.787,E2 -29805.787} C_VEL
LIN {X 0,Y 76.268,Z 310.277,A -85,B 0,C 180,E1 -29817.435,E2 -29817.435} C_VEL
LIN {X 0,Y 75.909,Z 306.412,A -85,B 0,C 180,E1 -29828.147,E2 -29828.147} C_VEL
LIN {X 0,Y 77.713,Z 302.4,A -85,B 0,C 180,E1 -29836.342,E2 -29836.342} C_VEL
LIN {X 0,Y 79.865,Z 298.737,A -85,B 0,C 180,E1 -29842.37,E2 -29842.37} C_VEL
LIN {X 0,Y 81.649,Z 294.856,A -85,B 0,C 180,E1 -29848.537,E2 -29848.537} C_VEL
LIN {X 0,Y 82.032,Z 293.524,A -85,B 0,C 180,E1 -29851.099,E2 -29851.099} C_VEL
LIN {X 0,Y 81.67,Z 292.103,A -85,B 0,C 180,E1 -29855.118,E2 -29855.118} C_VEL
LIN {X 0,Y 80.709,Z 291.256,A -85,B 0,C 180,E1 -29859.243,E2 -29859.243} C_VEL
LIN {X 0,Y 78.896,Z 289.712,A -85,B 0,C 180,E1 -29871.087,E2 -29871.087} C_VEL
LIN {X 0,Y 79.374,Z 288.995,A -85,B 0,C 180,E1 -29874.923,E2 -29874.923} C_VEL
LIN {X 0,Y 80.132,Z 288.37,A -85,B 0,C 180,E1 -29880.003,E2 -29880.003} C_VEL
LIN {X 0,Y 79.513,Z 289.304,A -85,B 0,C 180,E1 -29885.074,E2 -29885.074} C_VEL
LIN {X 0,Y 78.735,Z 291.017,A -85,B 0,C 180,E1 -29890.93,E2 -29890.93} C_VEL
LIN {X 0,Y 77.445,Z 293.374,A -85,B 0,C 180,E1 -29895.801,E2 -29895.801} C_VEL
LIN {X 0,Y 76.815,Z 294.447,A -85,B 0,C 180,E1 -29897.635,E2 -29897.635} C_VEL
LIN {X 0,Y 73.479,Z 297.649,A -85,B 0,C 180,E1 -29901.167,E2 -29901.167} C_VEL
LIN {X 0,Y 72.086,Z 298.818,A -85,B 0,C 180,E1 -29902.153,E2 -29902.153} C_VEL
LIN {X 0,Y 63.038,Z 304.845,A -85,B 0,C 180,E1 -29906.888,E2 -29906.888} C_VEL
LIN {X 0,Y 54.497,Z 309.595,A -85,B 0,C 180,E1 -29913.045,E2 -29913.045} C_VEL
LIN {X 0,Y 46.798,Z 313.211,A -85,B 0,C 180,E1 -29921.334,E2 -29921.334} C_VEL
LIN {X 0,Y 42.312,Z 315.016,A -85,B 0,C 180,E1 -29928.365,E2 -29928.365} C_VEL
LIN {X 0,Y 36.014,Z 317.486,A -85,B 0,C 180,E1 -29947.027,E2 -29947.027} C_VEL
LIN {X 0,Y 34.491,Z 318.087,A -85,B 0,C 180,E1 -29958.243,E2 -29958.243} C_VEL
LIN {X 0,Y 34.245,Z 318.254,A -85,B 0,C 180,E1 -29970,E2 -29970} C_VEL
LIN {X 0,Y 34.491,Z 318.087,A -85,B 0,C 180,E1 -29981.757,E2 -29981.757} C_VEL
LIN {X 0,Y 36.014,Z 317.486,A -85,B 0,C 180,E1 -29992.972,E2 -29992.972} C_VEL
LIN {X 0,Y 42.312,Z 315.016,A -85,B 0,C 180,E1 -30011.635,E2 -30011.635} C_VEL
LIN {X 0,Y 49.255,Z 312.058,A -85,B 0,C 180,E1 -30021.698,E2 -30021.698} C_VEL
LIN {X 0,Y 57.288,Z 308.064,A -85,B 0,C 180,E1 -30029.176,E2 -30029.176} C_VEL
LIN {X 0,Y 65.931,Z 302.984,A -85,B 0,C 180,E1 -30034.758,E2 -30034.758} C_VEL
LIN {X 0,Y 72.068,Z 298.816,A -85,B 0,C 180,E1 -30037.883,E2 -30037.883} C_VEL
LIN {X 0,Y 74.752,Z 296.467,A -85,B 0,C 180,E1 -30040.079,E2 -30040.079} C_VEL
LIN {X 0,Y 76.822,Z 294.444,A -85,B 0,C 180,E1 -30042.361,E2 -30042.361} C_VEL
LIN {X 0,Y 78.357,Z 291.76,A -85,B 0,C 180,E1 -30047.303,E2 -30047.303} C_VEL
LIN {X 0,Y 78.824,Z 290.794,A -85,B 0,C 180,E1 -30049.725,E2 -30049.725} C_VEL
LIN {X 0,Y 79.53,Z 289.291,A -85,B 0,C 180,E1 -30054.927,E2 -30054.927} C_VEL
LIN {X 0,Y 80.117,Z 288.381,A -85,B 0,C 180,E1 -30059.997,E2 -30059.997} C_VEL
LIN {X 0,Y 79.073,Z 289.381,A -85,B 0,C 180,E1 -30067.137,E2 -30067.137} C_VEL
LIN {X 0,Y 78.749,Z 290.126,A -85,B 0,C 180,E1 -30070.981,E2 -30070.981} C_VEL
LIN {X 0,Y 78.098,Z 292.322,A -85,B 0,C 180,E1 -30078.356,E2 -30078.356} C_VEL
LIN {X 0,Y 76.931,Z 294.778,A -85,B 0,C 180,E1 -30084.002,E2 -30084.002} C_VEL
LIN {X 0,Y 75.601,Z 297.643,A -85,B 0,C 180,E1 -30089.781,E2 -30089.781} C_VEL
LIN {X 0,Y 73.899,Z 300.321,A -85,B 0,C 180,E1 -30094.79,E2 -30094.79} C_VEL
LIN {X 0,Y 71.25,Z 304.122,A -85,B 0,C 180,E1 -30102,E2 -30102} C_VEL
LIN {X 0,Y 69.421,Z 307.155,A -85,B 0,C 180,E1 -30108.85,E2 -30108.85} C_VEL
LIN {X 0,Y 68.88,Z 310.528,A -85,B 0,C 180,E1 -30119.326,E2 -30119.326} C_VEL
LIN {X 0,Y 69.963,Z 312.168,A -85,B 0,C 180,E1 -30126.309,E2 -30126.309} C_VEL
LIN {X 0,Y 75.755,Z 314.284,A -85,B 0,C 180,E1 -30139.307,E2 -30139.307} C_VEL
LIN {X 0,Y 84.345,Z 314.725,A -85,B 0,C 180,E1 -30149,E2 -30149} C_VEL
LIN {X 0,Y 85.532,Z 314.689,A -85,B 0,C 180,E1 -30150,E2 -30150} C_VEL
LIN {X 0,Y 77.981,Z 314.514,A -85,B 0,C 180,E1 -30157.558,E2 -30157.558} C_VEL
LIN {X 0,Y 72.295,Z 313.392,A -85,B 0,C 180,E1 -30166.956,E2 -30166.956} C_VEL
LIN {X 0,Y 69.704,Z 311.892,A -85,B 0,C 180,E1 -30174.855,E2 -30174.855} C_VEL
LIN {X 0,Y 68.778,Z 309.144,A -85,B 0,C 180,E1 -30185.173,E2 -30185.173} C_VEL
LIN {X 0,Y 70.151,Z 305.702,A -85,B 0,C 180,E1 -30194.53,E2 -30194.53} C_VEL
LIN {X 0,Y 73.111,Z 301.482,A -85,B 0,C 180,E1 -30203.082,E2 -30203.082} C_VEL
LIN {X 0,Y 74.795,Z 299,A -85,B 0,C 180,E1 -30207.742,E2 -30207.742} C_VEL
LIN {X 0,Y 76.136,Z 296.453,A -85,B 0,C 180,E1 -30212.517,E2 -30212.517} C_VEL
LIN {X 0,Y 77.556,Z 293.56,A -85,B 0,C 180,E1 -30218.751,E2 -30218.751} C_VEL
LIN {X 0,Y 78.069,Z 292.346,A -85,B 0,C 180,E1 -30221.637,E2 -30221.637} C_VEL
LIN {X 0,Y 78.813,Z 289.964,A -85,B 0,C 180,E1 -30229.729,E2 -30229.729} C_VEL
LIN {X 0,Y 78.896,Z 289.712,A -85,B 0,C 180,E1 -30231.087,E2 -30231.087} C_VEL
LIN {X 0,Y 78.624,Z 289.657,A -85,B 0,C 180,E1 -30233.919,E2 -30233.919} C_VEL
LIN {X 0,Y 77.672,Z 290.296,A -85,B 0,C 180,E1 -30236.701,E2 -30236.701} C_VEL
LIN {X 0,Y 73.487,Z 294.094,A -85,B 0,C 180,E1 -30246.279,E2 -30246.279} C_VEL
LIN {X 0,Y 72.592,Z 295.513,A -85,B 0,C 180,E1 -30251.168,E2 -30251.168} C_VEL
LIN {X 0,Y 71.542,Z 296.839,A -85,B 0,C 180,E1 -30254.217,E2 -30254.217} C_VEL
LIN {X 0,Y 69.577,Z 298.591,A -85,B 0,C 180,E1 -30256.344,E2 -30256.344} C_VEL
LIN {X 0,Y 68.086,Z 299.76,A -85,B 0,C 180,E1 -30257.294,E2 -30257.294} C_VEL
LIN {X 0,Y 57.053,Z 306.296,A -85,B 0,C 180,E1 -30262.503,E2 -30262.503} C_VEL
LIN {X 0,Y 48.033,Z 310.626,A -85,B 0,C 180,E1 -30268.613,E2 -30268.613} C_VEL
LIN {X 0,Y 42.423,Z 312.999,A -85,B 0,C 180,E1 -30274.074,E2 -30274.074} C_VEL
LIN {X 0,Y 37.282,Z 314.804,A -85,B 0,C 180,E1 -30281.059,E2 -30281.059} C_VEL
LIN {X 0,Y 29.596,Z 317.274,A -85,B 0,C 180,E1 -30301.645,E2 -30301.645} C_VEL
LIN {X 0,Y 27.56,Z 317.875,A -85,B 0,C 180,E1 -30315.226,E2 -30315.226} C_VEL
LIN {X 0,Y 27.132,Z 318.042,A -85,B 0,C 180,E1 -30330,E2 -30330} C_VEL
LIN {X 0,Y 27.56,Z 317.875,A -85,B 0,C 180,E1 -30344.774,E2 -30344.774} C_VEL
LIN {X 0,Y 29.596,Z 317.274,A -85,B 0,C 180,E1 -30358.354,E2 -30358.354} C_VEL
LIN {X 0,Y 37.282,Z 314.804,A -85,B 0,C 180,E1 -30378.941,E2 -30378.941} C_VEL
LIN {X 0,Y 45.186,Z 311.846,A -85,B 0,C 180,E1 -30388.808,E2 -30388.808} C_VEL
LIN {X 0,Y 53.988,Z 307.852,A -85,B 0,C 180,E1 -30395.674,E2 -30395.674} C_VEL
LIN {X 0,Y 63.522,Z 302.587,A -85,B 0,C 180,E1 -30400.761,E2 -30400.761} C_VEL
LIN {X 0,Y 68.079,Z 299.759,A -85,B 0,C 180,E1 -30402.725,E2 -30402.725} C_VEL
LIN {X 0,Y 69.578,Z 298.592,A -85,B 0,C 180,E1 -30403.652,E2 -30403.652} C_VEL
LIN {X 0,Y 71.549,Z 296.835,A -85,B 0,C 180,E1 -30405.784,E2 -30405.784} C_VEL
LIN {X 0,Y 72.614,Z 295.499,A -85,B 0,C 180,E1 -30408.836,E2 -30408.836} C_VEL
